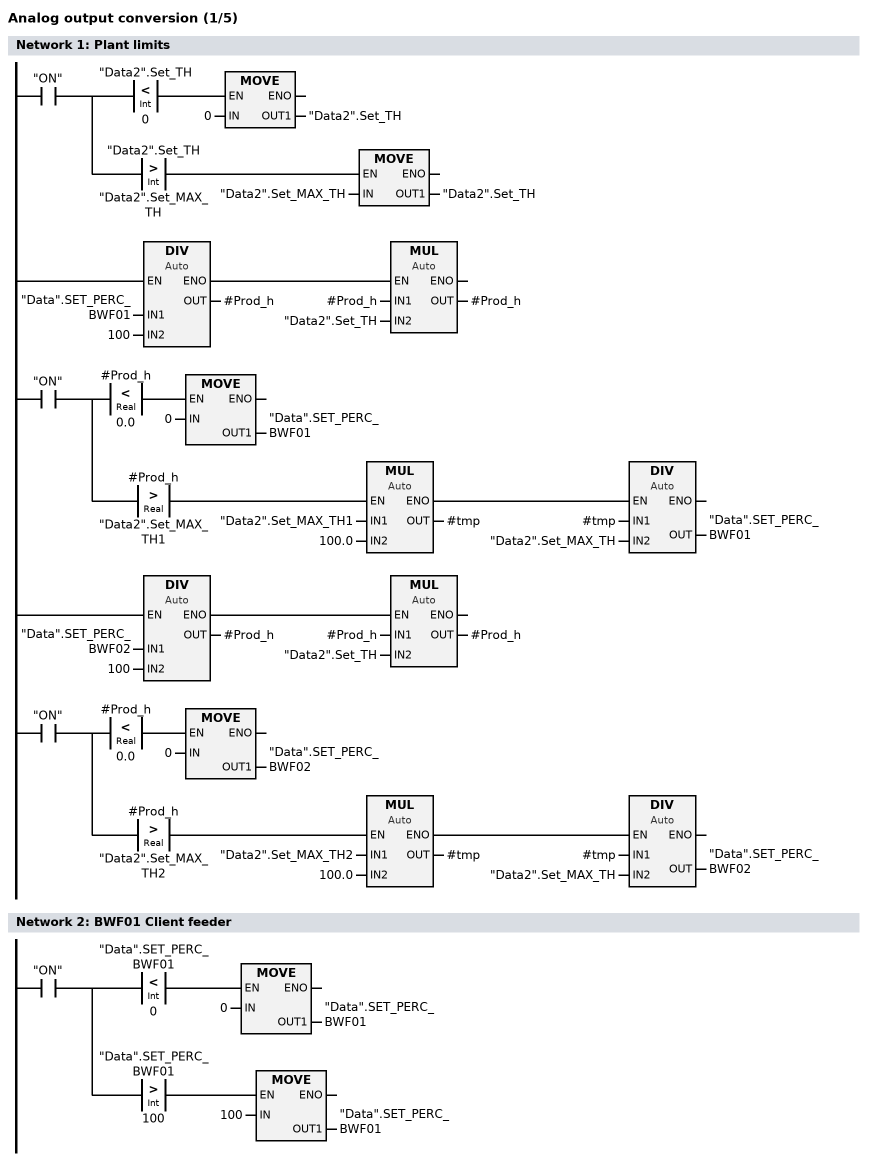
   RUNG wire#powerrail
      Contact( "ON" )
      wire#w1
      { S7_Templates := "SrcType := Int" } LT_Contact(in1 := "Data2".Set_TH, in2 := 0)
      { S7_GenerateENO := "TRUE" } Move(in := 0, out1 => "Data2".Set_TH)
   END_RUNG
   RUNG wire#w1
      { S7_Templates := "SrcType := Int" } GT_Contact(in1 := "Data2".Set_TH, in2 := "Data2".Set_MAX_TH)
      { S7_GenerateENO := "TRUE" } Move(in := "Data2".Set_MAX_TH, out1 => "Data2".Set_TH)
   END_RUNG
   RUNG wire#powerrail
      Div(in1 := "Data".SET_PERC_BWF01, in2 := 100, out => #Prod_h)
      Mul(in1 := #Prod_h, in2 := "Data2".Set_TH, out => #Prod_h)
   END_RUNG
   RUNG wire#powerrail
      Contact( "ON" )
      wire#w2
      { S7_Templates := "SrcType := Real" } LT_Contact(in1 := #Prod_h, in2 := 0.0)
      { S7_GenerateENO := "TRUE" } Move(in := 0, out1 => "Data".SET_PERC_BWF01)
   END_RUNG
   RUNG wire#w2
      { S7_Templates := "SrcType := Real" } GT_Contact(in1 := #Prod_h, in2 := "Data2".Set_MAX_TH1)
      Mul(in1 := "Data2".Set_MAX_TH1, in2 := 100.0, out => #tmp)
      Div(in1 := #tmp, in2 := "Data2".Set_MAX_TH, out => "Data".SET_PERC_BWF01)
   END_RUNG
   RUNG wire#powerrail
      Div(in1 := "Data".SET_PERC_BWF02, in2 := 100, out => #Prod_h)
      Mul(in1 := #Prod_h, in2 := "Data2".Set_TH, out => #Prod_h)
   END_RUNG
   RUNG wire#powerrail
      Contact( "ON" )
      wire#w3
      { S7_Templates := "SrcType := Real" } LT_Contact(in1 := #Prod_h, in2 := 0.0)
      { S7_GenerateENO := "TRUE" } Move(in := 0, out1 => "Data".SET_PERC_BWF02)
   END_RUNG
   RUNG wire#w3
      { S7_Templates := "SrcType := Real" } GT_Contact(in1 := #Prod_h, in2 := "Data2".Set_MAX_TH2)
      Mul(in1 := "Data2".Set_MAX_TH2, in2 := 100.0, out => #tmp)
      Div(in1 := #tmp, in2 := "Data2".Set_MAX_TH, out => "Data".SET_PERC_BWF02)
   END_RUNG
   // the same network as SCL:
   IF "ON" AND ("Data2".Set_TH < 0) THEN "Data2".Set_TH := 0; END_IF;
   IF "ON" AND ("Data2".Set_TH > "Data2".Set_MAX_TH) THEN "Data2".Set_TH := "Data2".Set_MAX_TH; END_IF;
   #Prod_h := "Data".SET_PERC_BWF01 / 100;
   #Prod_h := #Prod_h * "Data2".Set_TH;
   IF "ON" AND (#Prod_h < 0.0) THEN "Data".SET_PERC_BWF01 := 0; END_IF;
   IF "ON" AND (#Prod_h > "Data2".Set_MAX_TH1) THEN
       #tmp := "Data2".Set_MAX_TH1 * 100.0;
       "Data".SET_PERC_BWF01 := #tmp / "Data2".Set_MAX_TH;
   END_IF;
   #Prod_h := "Data".SET_PERC_BWF02 / 100;
   #Prod_h := #Prod_h * "Data2".Set_TH;
   IF "ON" AND (#Prod_h < 0.0) THEN "Data".SET_PERC_BWF02 := 0; END_IF;
   IF "ON" AND (#Prod_h > "Data2".Set_MAX_TH2) THEN
       #tmp := "Data2".Set_MAX_TH2 * 100.0;
       "Data".SET_PERC_BWF02 := #tmp / "Data2".Set_MAX_TH;
   END_IF;
END_REGION

REGION Network 2: BWF01 Client feeder
   RUNG wire#powerrail
      Contact( "ON" )
      wire#w1
      { S7_Templates := "SrcType := Int" } LT_Contact(in1 := "Data".SET_PERC_BWF01, in2 := 0)
      { S7_GenerateENO := "TRUE" } Move(in := 0, out1 => "Data".SET_PERC_BWF01)
   END_RUNG
   RUNG wire#w1
      { S7_Templates := "SrcType := Int" } GT_Contact(in1 := "Data".SET_PERC_BWF01, in2 := 100)
      { S7_GenerateENO := "TRUE" } Move(in := 100, out1 => "Data".SET_PERC_BWF01)
   END_RUNG
   // the same network as SCL:
   IF "ON" AND ("Data".SET_PERC_BWF01 < 0) THEN "Data".SET_PERC_BWF01 := 0; END_IF;
   IF "ON" AND ("Data".SET_PERC_BWF01 > 100) THEN "Data".SET_PERC_BWF01 := 100; END_IF;
END_REGION

REGION Network 3: BWF01 speed calculation
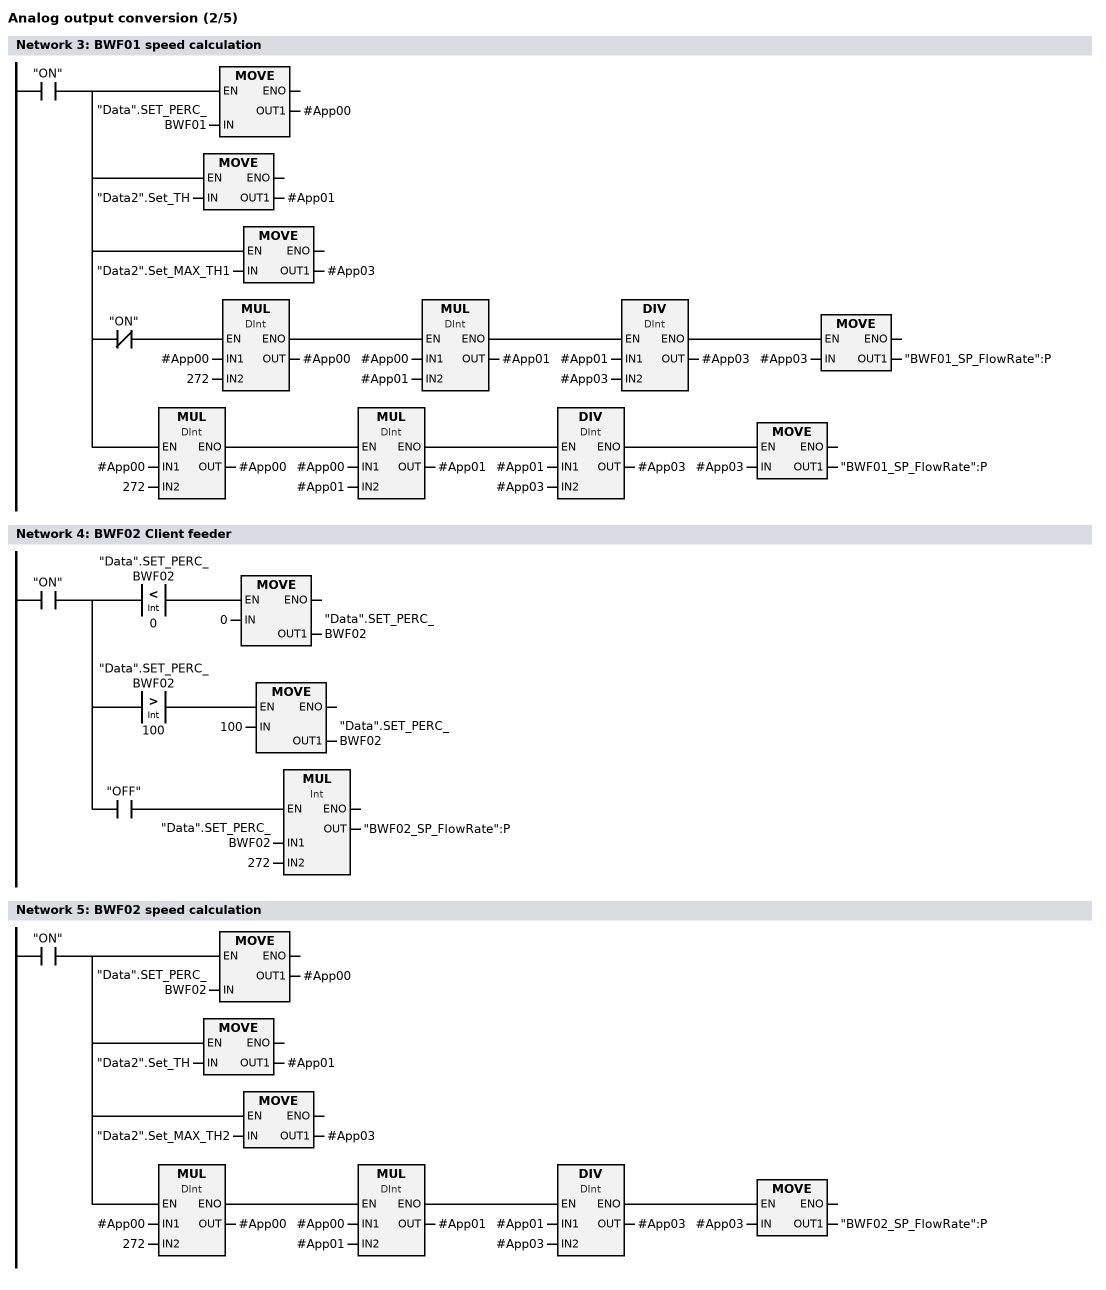
   RUNG wire#powerrail
      Contact( "ON" )
      wire#w1
      { S7_GenerateENO := "TRUE" } Move(in := "Data".SET_PERC_BWF01, out1 => #App00)
   END_RUNG
   RUNG wire#w1
      { S7_GenerateENO := "TRUE" } Move(in := "Data2".Set_TH, out1 => #App01)
   END_RUNG
   RUNG wire#w1
      { S7_GenerateENO := "TRUE" } Move(in := "Data2".Set_MAX_TH1, out1 => #App03)
   END_RUNG
   RUNG wire#w1
      I_Contact( "ON" )
      { S7_Templates := "SrcType := DInt"; S7_GenerateENO := "TRUE" } Mul(in1 := #App00, in2 := 272, out => #App00)
      { S7_Templates := "SrcType := DInt"; S7_GenerateENO := "TRUE" } Mul(in1 := #App00, in2 := #App01, out => #App01)
      { S7_Templates := "SrcType := DInt"; S7_GenerateENO := "TRUE" } Div(in1 := #App01, in2 := #App03, out => #App03)
      { S7_GenerateENO := "TRUE" } Move(in := #App03, out1 => "BWF01_SP_FlowRate":P)
   END_RUNG
   RUNG wire#w1
      { S7_Templates := "SrcType := DInt"; S7_GenerateENO := "TRUE" } Mul(in1 := #App00, in2 := 272, out => #App00)
      { S7_Templates := "SrcType := DInt"; S7_GenerateENO := "TRUE" } Mul(in1 := #App00, in2 := #App01, out => #App01)
      { S7_Templates := "SrcType := DInt"; S7_GenerateENO := "TRUE" } Div(in1 := #App01, in2 := #App03, out => #App03)
      { S7_GenerateENO := "TRUE" } Move(in := #App03, out1 => "BWF01_SP_FlowRate":P)
   END_RUNG
   // the same network as SCL:
   // ENO of a box is taken as its EN; it also drops when the box reports an error
   IF "ON" THEN
       #App00 := "Data".SET_PERC_BWF01;
       #App01 := "Data2".Set_TH;
       #App03 := "Data2".Set_MAX_TH1;
   END_IF;
   IF "ON" AND NOT "ON" THEN
       #App00 := #App00 * 272;
       #App01 := #App00 * #App01;
       #App03 := #App01 / #App03;
       "BWF01_SP_FlowRate":P := #App03;
   END_IF;
   IF "ON" THEN
       #App00 := #App00 * 272;
       #App01 := #App00 * #App01;
       #App03 := #App01 / #App03;
       "BWF01_SP_FlowRate":P := #App03;
   END_IF;
END_REGION

REGION Network 4: BWF02 Client feeder
   RUNG wire#powerrail
      Contact( "ON" )
      wire#w1
      { S7_Templates := "SrcType := Int" } LT_Contact(in1 := "Data".SET_PERC_BWF02, in2 := 0)
      { S7_GenerateENO := "TRUE" } Move(in := 0, out1 => "Data".SET_PERC_BWF02)
   END_RUNG
   RUNG wire#w1
      { S7_Templates := "SrcType := Int" } GT_Contact(in1 := "Data".SET_PERC_BWF02, in2 := 100)
      { S7_GenerateENO := "TRUE" } Move(in := 100, out1 => "Data".SET_PERC_BWF02)
   END_RUNG
   RUNG wire#w1
      Contact( "OFF" )
      { S7_Templates := "SrcType := Int"; S7_GenerateENO := "TRUE" } Mul(in1 := "Data".SET_PERC_BWF02, in2 := 272, out => "BWF02_SP_FlowRate":P)
   END_RUNG
   // the same network as SCL:
   IF "ON" AND ("Data".SET_PERC_BWF02 < 0) THEN "Data".SET_PERC_BWF02 := 0; END_IF;
   IF "ON" AND ("Data".SET_PERC_BWF02 > 100) THEN "Data".SET_PERC_BWF02 := 100; END_IF;
   IF "ON" AND "OFF" THEN "BWF02_SP_FlowRate":P := "Data".SET_PERC_BWF02 * 272; END_IF;
END_REGION

REGION Network 5: BWF02 speed calculation
   RUNG wire#powerrail
      Contact( "ON" )
      wire#w1
      { S7_GenerateENO := "TRUE" } Move(in := "Data".SET_PERC_BWF02, out1 => #App00)
   END_RUNG
   RUNG wire#w1
      { S7_GenerateENO := "TRUE" } Move(in := "Data2".Set_TH, out1 => #App01)
   END_RUNG
   RUNG wire#w1
      { S7_GenerateENO := "TRUE" } Move(in := "Data2".Set_MAX_TH2, out1 => #App03)
   END_RUNG
   RUNG wire#w1
      { S7_Templates := "SrcType := DInt"; S7_GenerateENO := "TRUE" } Mul(in1 := #App00, in2 := 272, out => #App00)
      { S7_Templates := "SrcType := DInt"; S7_GenerateENO := "TRUE" } Mul(in1 := #App00, in2 := #App01, out => #App01)
      { S7_Templates := "SrcType := DInt"; S7_GenerateENO := "TRUE" } Div(in1 := #App01, in2 := #App03, out => #App03)
      { S7_GenerateENO := "TRUE" } Move(in := #App03, out1 => "BWF02_SP_FlowRate":P)
   END_RUNG
   // the same network as SCL:
   // ENO of a box is taken as its EN; it also drops when the box reports an error
   IF "ON" THEN
       #App00 := "Data".SET_PERC_BWF02;
       #App01 := "Data2".Set_TH;
       #App03 := "Data2".Set_MAX_TH2;
       #App00 := #App00 * 272;
       #App01 := #App00 * #App01;
       #App03 := #App01 / #App03;
       "BWF02_SP_FlowRate":P := #App03;
   END_IF;
END_REGION

REGION Network 6: RD-01 Cylinder
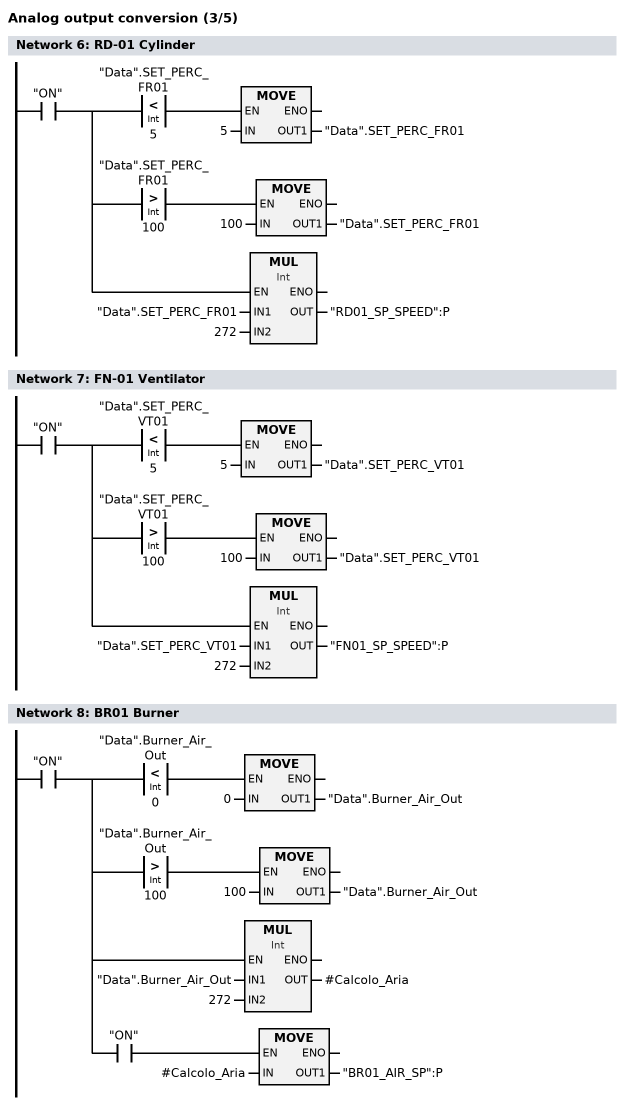
   RUNG wire#powerrail
      Contact( "ON" )
      wire#w1
      { S7_Templates := "SrcType := Int" } LT_Contact(in1 := "Data".SET_PERC_FR01, in2 := 5)
      { S7_GenerateENO := "TRUE" } Move(in := 5, out1 => "Data".SET_PERC_FR01)
   END_RUNG
   RUNG wire#w1
      { S7_Templates := "SrcType := Int" } GT_Contact(in1 := "Data".SET_PERC_FR01, in2 := 100)
      { S7_GenerateENO := "TRUE" } Move(in := 100, out1 => "Data".SET_PERC_FR01)
   END_RUNG
   RUNG wire#w1
      { S7_Templates := "SrcType := Int"; S7_GenerateENO := "TRUE" } Mul(in1 := "Data".SET_PERC_FR01, in2 := 272, out => "RD01_SP_SPEED":P)
   END_RUNG
   // the same network as SCL:
   IF "ON" AND ("Data".SET_PERC_FR01 < 5) THEN "Data".SET_PERC_FR01 := 5; END_IF;
   IF "ON" AND ("Data".SET_PERC_FR01 > 100) THEN "Data".SET_PERC_FR01 := 100; END_IF;
   IF "ON" THEN "RD01_SP_SPEED":P := "Data".SET_PERC_FR01 * 272; END_IF;
END_REGION

REGION Network 7: FN-01 Ventilator
   RUNG wire#powerrail
      Contact( "ON" )
      wire#w1
      { S7_Templates := "SrcType := Int" } LT_Contact(in1 := "Data".SET_PERC_VT01, in2 := 5)
      { S7_GenerateENO := "TRUE" } Move(in := 5, out1 => "Data".SET_PERC_VT01)
   END_RUNG
   RUNG wire#w1
      { S7_Templates := "SrcType := Int" } GT_Contact(in1 := "Data".SET_PERC_VT01, in2 := 100)
      { S7_GenerateENO := "TRUE" } Move(in := 100, out1 => "Data".SET_PERC_VT01)
   END_RUNG
   RUNG wire#w1
      { S7_Templates := "SrcType := Int"; S7_GenerateENO := "TRUE" } Mul(in1 := "Data".SET_PERC_VT01, in2 := 272, out => "FN01_SP_SPEED":P)
   END_RUNG
   // the same network as SCL:
   IF "ON" AND ("Data".SET_PERC_VT01 < 5) THEN "Data".SET_PERC_VT01 := 5; END_IF;
   IF "ON" AND ("Data".SET_PERC_VT01 > 100) THEN "Data".SET_PERC_VT01 := 100; END_IF;
   IF "ON" THEN "FN01_SP_SPEED":P := "Data".SET_PERC_VT01 * 272; END_IF;
END_REGION

REGION Network 8: BR01 Burner
   RUNG wire#powerrail
      Contact( "ON" )
      wire#w1
      { S7_Templates := "SrcType := Int" } LT_Contact(in1 := "Data".Burner_Air_Out, in2 := 0)
      { S7_GenerateENO := "TRUE" } Move(in := 0, out1 => "Data".Burner_Air_Out)
   END_RUNG
   RUNG wire#w1
      { S7_Templates := "SrcType := Int" } GT_Contact(in1 := "Data".Burner_Air_Out, in2 := 100)
      { S7_GenerateENO := "TRUE" } Move(in := 100, out1 => "Data".Burner_Air_Out)
   END_RUNG
   RUNG wire#w1
      { S7_Templates := "SrcType := Int"; S7_GenerateENO := "TRUE" } Mul(in1 := "Data".Burner_Air_Out, in2 := 272, out => #Calcolo_Aria)
   END_RUNG
   RUNG wire#w1
      Contact( "ON" )
      { S7_GenerateENO := "TRUE" } Move(in := #Calcolo_Aria, out1 => "BR01_AIR_SP":P)
   END_RUNG
   // the same network as SCL:
   IF "ON" AND ("Data".Burner_Air_Out < 0) THEN "Data".Burner_Air_Out := 0; END_IF;
   IF "ON" AND ("Data".Burner_Air_Out > 100) THEN "Data".Burner_Air_Out := 100; END_IF;
   IF "ON" THEN #Calcolo_Aria := "Data".Burner_Air_Out * 272; END_IF;
   IF "ON" AND "ON" THEN "BR01_AIR_SP":P := #Calcolo_Aria; END_IF;
END_REGION

REGION Network 9: BR01 Burner - Gas
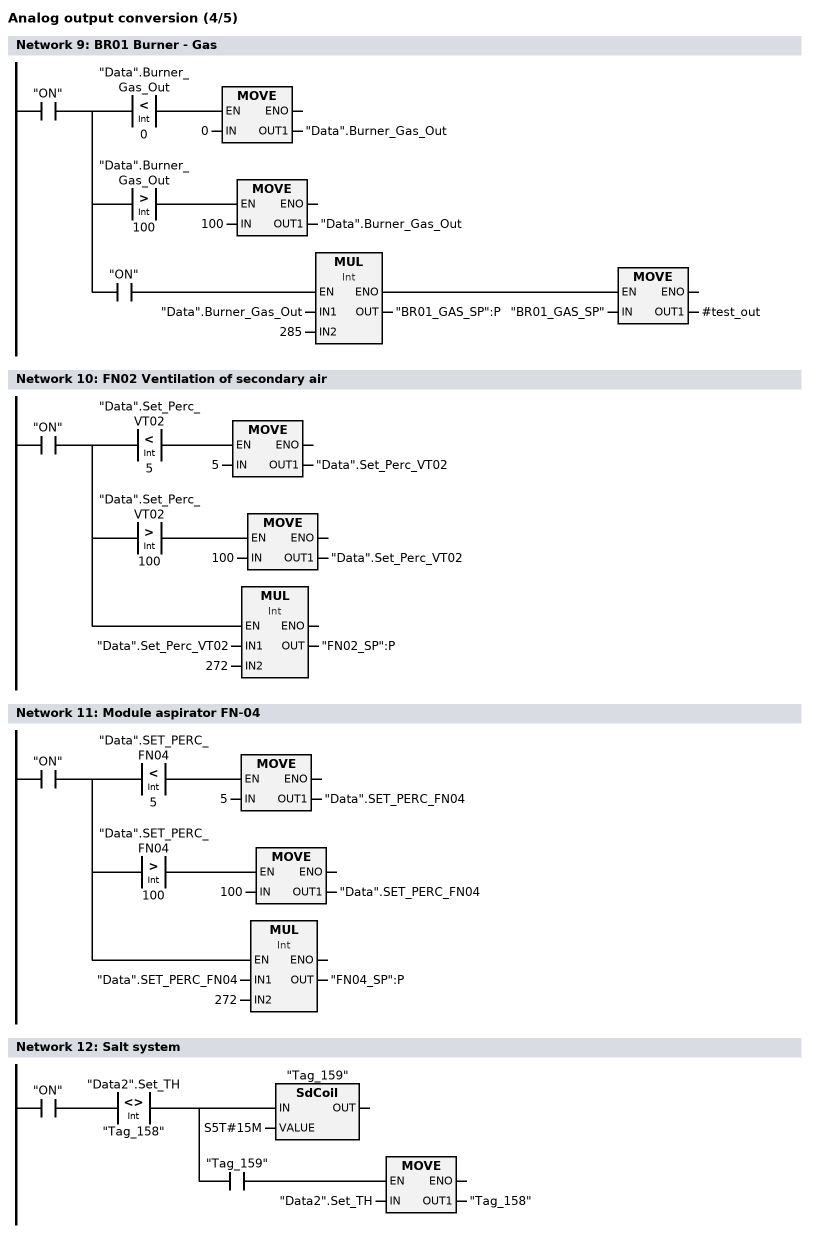
   RUNG wire#powerrail
      Contact( "ON" )
      wire#w1
      { S7_Templates := "SrcType := Int" } LT_Contact(in1 := "Data".Burner_Gas_Out, in2 := 0)
      { S7_GenerateENO := "TRUE" } Move(in := 0, out1 => "Data".Burner_Gas_Out)
   END_RUNG
   RUNG wire#w1
      { S7_Templates := "SrcType := Int" } GT_Contact(in1 := "Data".Burner_Gas_Out, in2 := 100)
      { S7_GenerateENO := "TRUE" } Move(in := 100, out1 => "Data".Burner_Gas_Out)
   END_RUNG
   RUNG wire#w1
      Contact( "ON" )
      { S7_Templates := "SrcType := Int"; S7_GenerateENO := "TRUE" } Mul(in1 := "Data".Burner_Gas_Out, in2 := 285, out => "BR01_GAS_SP":P)
      Move(in := "BR01_GAS_SP", out1 => #test_out)
   END_RUNG
   // the same network as SCL:
   // ENO of a box is taken as its EN; it also drops when the box reports an error
   IF "ON" AND ("Data".Burner_Gas_Out < 0) THEN "Data".Burner_Gas_Out := 0; END_IF;
   IF "ON" AND ("Data".Burner_Gas_Out > 100) THEN "Data".Burner_Gas_Out := 100; END_IF;
   IF "ON" AND "ON" THEN
       "BR01_GAS_SP":P := "Data".Burner_Gas_Out * 285;
       #test_out := "BR01_GAS_SP";
   END_IF;
END_REGION

REGION Network 10: FN02 Ventilation of secondary air
   RUNG wire#powerrail
      Contact( "ON" )
      wire#w1
      { S7_Templates := "SrcType := Int" } LT_Contact(in1 := "Data".Set_Perc_VT02, in2 := 5)
      { S7_GenerateENO := "TRUE" } Move(in := 5, out1 => "Data".Set_Perc_VT02)
   END_RUNG
   RUNG wire#w1
      { S7_Templates := "SrcType := Int" } GT_Contact(in1 := "Data".Set_Perc_VT02, in2 := 100)
      { S7_GenerateENO := "TRUE" } Move(in := 100, out1 => "Data".Set_Perc_VT02)
   END_RUNG
   RUNG wire#w1
      { S7_Templates := "SrcType := Int"; S7_GenerateENO := "TRUE" } Mul(in1 := "Data".Set_Perc_VT02, in2 := 272, out => "FN02_SP":P)
   END_RUNG
   // the same network as SCL:
   IF "ON" AND ("Data".Set_Perc_VT02 < 5) THEN "Data".Set_Perc_VT02 := 5; END_IF;
   IF "ON" AND ("Data".Set_Perc_VT02 > 100) THEN "Data".Set_Perc_VT02 := 100; END_IF;
   IF "ON" THEN "FN02_SP":P := "Data".Set_Perc_VT02 * 272; END_IF;
END_REGION

REGION Network 11: Module aspirator FN-04
   RUNG wire#powerrail
      Contact( "ON" )
      wire#w1
      { S7_Templates := "SrcType := Int" } LT_Contact(in1 := "Data".SET_PERC_FN04, in2 := 5)
      { S7_GenerateENO := "TRUE" } Move(in := 5, out1 => "Data".SET_PERC_FN04)
   END_RUNG
   RUNG wire#w1
      { S7_Templates := "SrcType := Int" } GT_Contact(in1 := "Data".SET_PERC_FN04, in2 := 100)
      { S7_GenerateENO := "TRUE" } Move(in := 100, out1 => "Data".SET_PERC_FN04)
   END_RUNG
   RUNG wire#w1
      { S7_Templates := "SrcType := Int"; S7_GenerateENO := "TRUE" } Mul(in1 := "Data".SET_PERC_FN04, in2 := 272, out => "FN04_SP":P)
   END_RUNG
   // the same network as SCL:
   IF "ON" AND ("Data".SET_PERC_FN04 < 5) THEN "Data".SET_PERC_FN04 := 5; END_IF;
   IF "ON" AND ("Data".SET_PERC_FN04 > 100) THEN "Data".SET_PERC_FN04 := 100; END_IF;
   IF "ON" THEN "FN04_SP":P := "Data".SET_PERC_FN04 * 272; END_IF;
END_REGION

REGION Network 12: Salt system
   // no SCL statement known for SdCoil: written as a call
   #_w1 := "ON" AND ("Data2".Set_TH <> "Tag_158");
   SdCoil(in := #_w1, value := S5T#15M, operand := "Tag_159");
   IF #_w1 AND "Tag_159" THEN "Tag_158" := "Data2".Set_TH; END_IF;
END_REGION

REGION Network 13: Send output to perifery
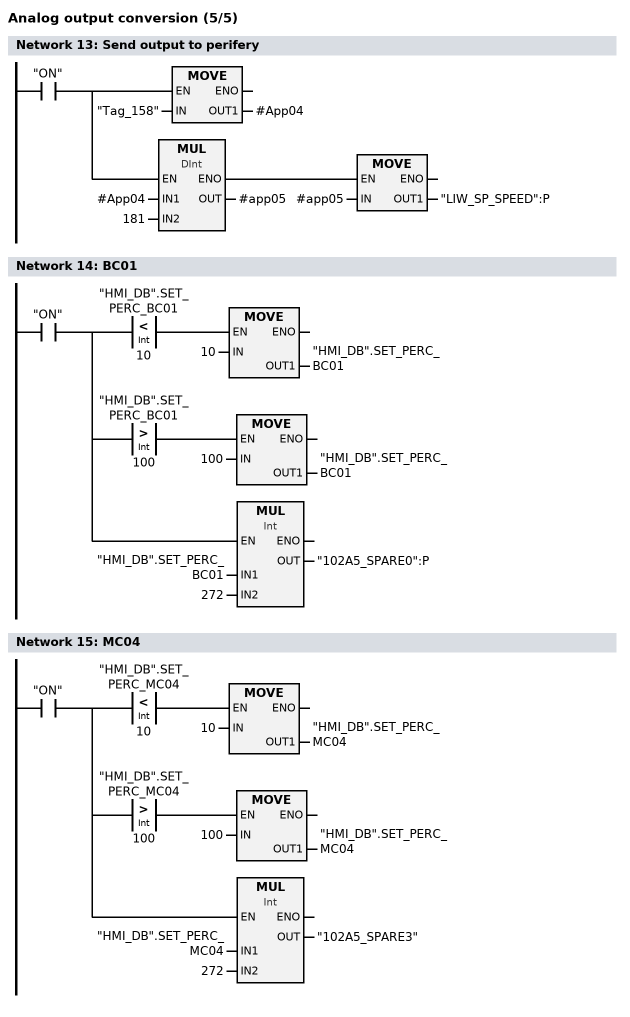
   RUNG wire#powerrail
      Contact( "ON" )
      wire#w1
      { S7_GenerateENO := "TRUE" } Move(in := "Tag_158", out1 => #App04)
   END_RUNG
   RUNG wire#w1
      { S7_Templates := "SrcType := DInt"; S7_GenerateENO := "TRUE" } Mul(in1 := #App04, in2 := 181, out => #app05)
      { S7_GenerateENO := "TRUE" } Move(in := #app05, out1 => "LIW_SP_SPEED":P)
   END_RUNG
   // the same network as SCL:
   // ENO of a box is taken as its EN; it also drops when the box reports an error
   IF "ON" THEN
       #App04 := "Tag_158";
       #app05 := #App04 * 181;
       "LIW_SP_SPEED":P := #app05;
   END_IF;
END_REGION

REGION Network 14: BC01
   RUNG wire#powerrail
      Contact( "ON" )
      wire#w1
      { S7_Templates := "SrcType := Int" } LT_Contact(in1 := "HMI_DB".SET_PERC_BC01, in2 := 10)
      { S7_GenerateENO := "TRUE" } Move(in := 10, out1 => "HMI_DB".SET_PERC_BC01)
   END_RUNG
   RUNG wire#w1
      { S7_Templates := "SrcType := Int" } GT_Contact(in1 := "HMI_DB".SET_PERC_BC01, in2 := 100)
      { S7_GenerateENO := "TRUE" } Move(in := 100, out1 => "HMI_DB".SET_PERC_BC01)
   END_RUNG
   RUNG wire#w1
      { S7_Templates := "SrcType := Int"; S7_GenerateENO := "TRUE" } Mul(in1 := "HMI_DB".SET_PERC_BC01, in2 := 272, out => "102A5_SPARE0":P)
   END_RUNG
   // the same network as SCL:
   IF "ON" AND ("HMI_DB".SET_PERC_BC01 < 10) THEN "HMI_DB".SET_PERC_BC01 := 10; END_IF;
   IF "ON" AND ("HMI_DB".SET_PERC_BC01 > 100) THEN "HMI_DB".SET_PERC_BC01 := 100; END_IF;
   IF "ON" THEN "102A5_SPARE0":P := "HMI_DB".SET_PERC_BC01 * 272; END_IF;
END_REGION

REGION Network 15: MC04
   RUNG wire#powerrail
      Contact( "ON" )
      wire#w1
      { S7_Templates := "SrcType := Int" } LT_Contact(in1 := "HMI_DB".SET_PERC_MC04, in2 := 10)
      { S7_GenerateENO := "TRUE" } Move(in := 10, out1 => "HMI_DB".SET_PERC_MC04)
   END_RUNG
   RUNG wire#w1
      { S7_Templates := "SrcType := Int" } GT_Contact(in1 := "HMI_DB".SET_PERC_MC04, in2 := 100)
      { S7_GenerateENO := "TRUE" } Move(in := 100, out1 => "HMI_DB".SET_PERC_MC04)
   END_RUNG
   RUNG wire#w1
      { S7_Templates := "SrcType := Int"; S7_GenerateENO := "TRUE" } Mul(in1 := "HMI_DB".SET_PERC_MC04, in2 := 272, out => "102A5_SPARE3")
   END_RUNG
   // the same network as SCL:
   IF "ON" AND ("HMI_DB".SET_PERC_MC04 < 10) THEN "HMI_DB".SET_PERC_MC04 := 10; END_IF;
   IF "ON" AND ("HMI_DB".SET_PERC_MC04 > 100) THEN "HMI_DB".SET_PERC_MC04 := 100; END_IF;
   IF "ON" THEN "102A5_SPARE3" := "HMI_DB".SET_PERC_MC04 * 272; END_IF;
END_REGION
END_FUNCTION

FUNCTION "Simulation" : Void   // FC20, LAD
{ S7_Optimized_Access := 'TRUE' }
VERSION : 0.1
   VAR_TEMP
      BuffInc : Int;
   END_VAR
BEGIN

REGION Network 1
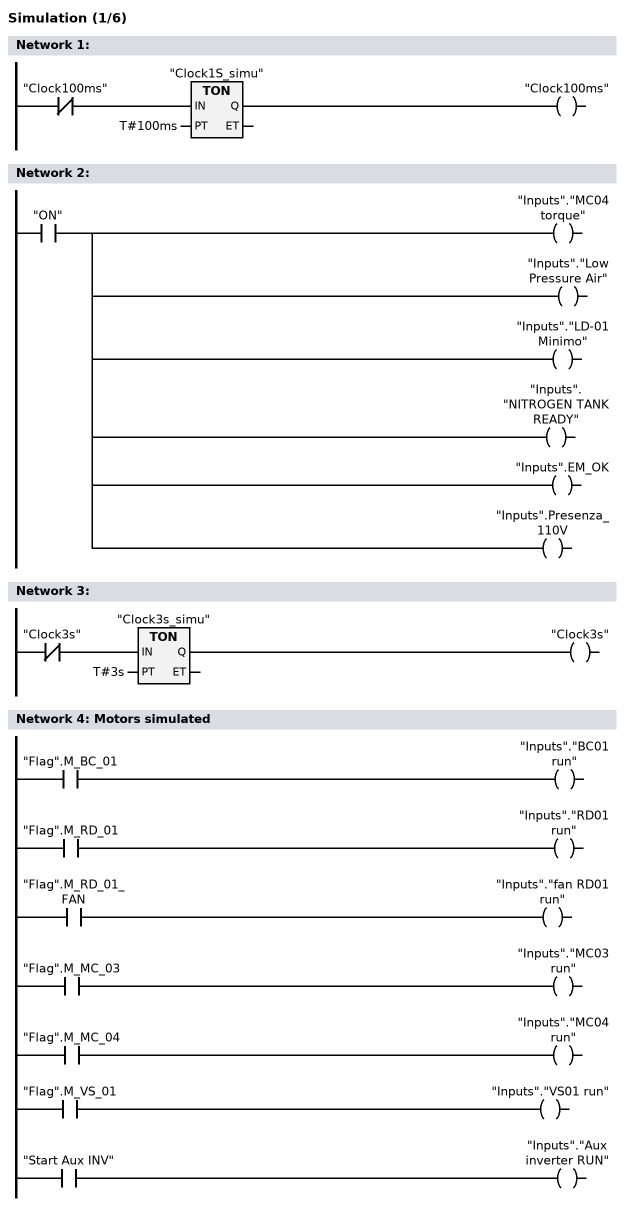
   "Clock1S_simu".TON(IN := NOT "Clock100ms", PT := T#100ms);
   "Clock100ms" := "Clock1S_simu".Q;
END_REGION

REGION Network 2
   RUNG wire#powerrail
      Contact( "ON" )
      wire#w1
      Coil( "Inputs"."MC04 torque" )
   END_RUNG
   RUNG wire#w1
      Coil( "Inputs"."Low Pressure Air" )
   END_RUNG
   RUNG wire#w1
      Coil( "Inputs"."LD-01 Minimo" )
   END_RUNG
   RUNG wire#w1
      Coil( "Inputs"."NITROGEN TANK READY" )
   END_RUNG
   RUNG wire#w1
      Coil( "Inputs".EM_OK )
   END_RUNG
   RUNG wire#w1
      Coil( "Inputs".Presenza_110V )
   END_RUNG
   // the same network as SCL:
   "Inputs"."MC04 torque" := "ON";
   "Inputs"."Low Pressure Air" := "ON";
   "Inputs"."LD-01 Minimo" := "ON";
   "Inputs"."NITROGEN TANK READY" := "ON";
   "Inputs".EM_OK := "ON";
   "Inputs".Presenza_110V := "ON";
END_REGION

REGION Network 3
   "Clock3s_simu".TON(IN := NOT "Clock3s", PT := T#3s);
   "Clock3s" := "Clock3s_simu".Q;
END_REGION

REGION Network 4: Motors simulated
   RUNG wire#powerrail
      Contact( "Flag".M_BC_01 )
      Coil( "Inputs"."BC01 run" )
   END_RUNG
   RUNG wire#powerrail
      Contact( "Flag".M_RD_01 )
      Coil( "Inputs"."RD01 run" )
   END_RUNG
   RUNG wire#powerrail
      Contact( "Flag".M_RD_01_FAN )
      Coil( "Inputs"."fan RD01 run" )
   END_RUNG
   RUNG wire#powerrail
      Contact( "Flag".M_MC_03 )
      Coil( "Inputs"."MC03 run" )
   END_RUNG
   RUNG wire#powerrail
      Contact( "Flag".M_MC_04 )
      Coil( "Inputs"."MC04 run" )
   END_RUNG
   RUNG wire#powerrail
      Contact( "Flag".M_VS_01 )
      Coil( "Inputs"."VS01 run" )
   END_RUNG
   RUNG wire#powerrail
      Contact( "Start Aux INV" )
      Coil( "Inputs"."Aux inverter RUN" )
   END_RUNG
   // the same network as SCL:
   "Inputs"."BC01 run" := "Flag".M_BC_01;
   "Inputs"."RD01 run" := "Flag".M_RD_01;
   "Inputs"."fan RD01 run" := "Flag".M_RD_01_FAN;
   "Inputs"."MC03 run" := "Flag".M_MC_03;
   "Inputs"."MC04 run" := "Flag".M_MC_04;
   "Inputs"."VS01 run" := "Flag".M_VS_01;
   "Inputs"."Aux inverter RUN" := "Start Aux INV";
END_REGION

REGION Network 5: MV
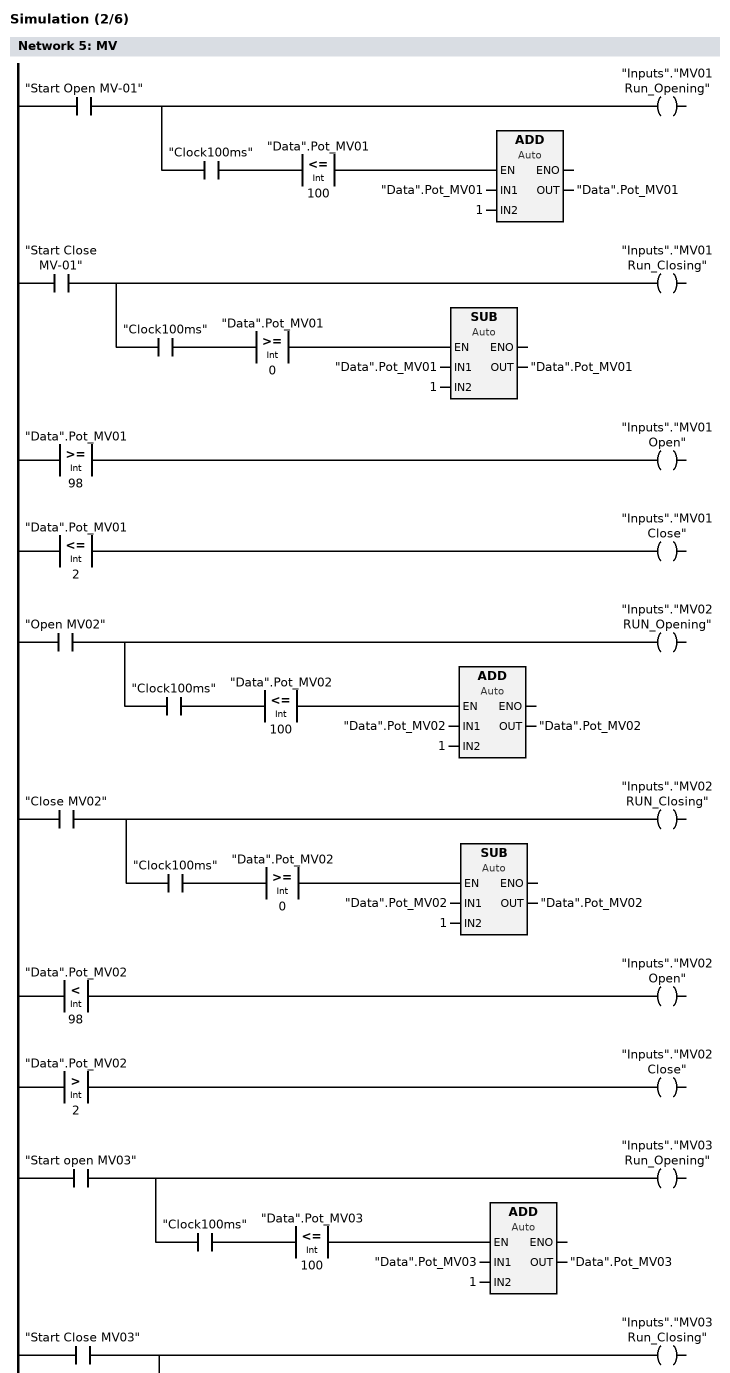
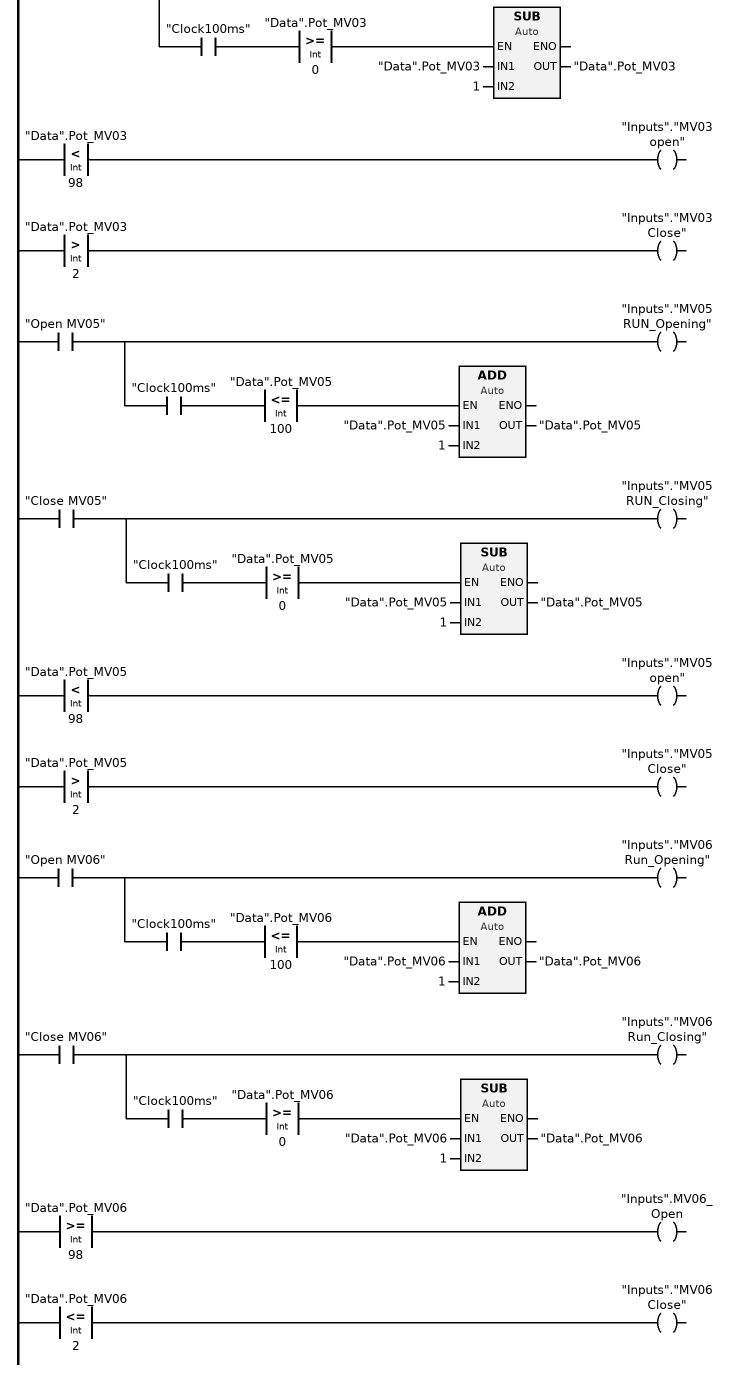
   RUNG wire#powerrail
      Contact( "Start Open MV-01" )
      wire#w1
      Coil( "Inputs"."MV01 Run_Opening" )
   END_RUNG
   RUNG wire#w1
      Contact( "Clock100ms" )
      { S7_Templates := "SrcType := Int" } LE_Contact(in1 := "Data".Pot_MV01, in2 := 100)
      Add(in1 := "Data".Pot_MV01, in2 := 1, out => "Data".Pot_MV01)
   END_RUNG
   RUNG wire#powerrail
      Contact( "Start Close MV-01" )
      wire#w2
      Coil( "Inputs"."MV01 Run_Closing" )
   END_RUNG
   RUNG wire#w2
      Contact( "Clock100ms" )
      { S7_Templates := "SrcType := Int" } GE_Contact(in1 := "Data".Pot_MV01, in2 := 0)
      Sub(in1 := "Data".Pot_MV01, in2 := 1, out => "Data".Pot_MV01)
   END_RUNG
   RUNG wire#powerrail
      { S7_Templates := "SrcType := Int" } GE_Contact(in1 := "Data".Pot_MV01, in2 := 98)
      Coil( "Inputs"."MV01 Open" )
   END_RUNG
   RUNG wire#powerrail
      { S7_Templates := "SrcType := Int" } LE_Contact(in1 := "Data".Pot_MV01, in2 := 2)
      Coil( "Inputs"."MV01 Close" )
   END_RUNG
   RUNG wire#powerrail
      Contact( "Open MV02" )
      wire#w3
      Coil( "Inputs"."MV02 RUN_Opening" )
   END_RUNG
   RUNG wire#w3
      Contact( "Clock100ms" )
      { S7_Templates := "SrcType := Int" } LE_Contact(in1 := "Data".Pot_MV02, in2 := 100)
      Add(in1 := "Data".Pot_MV02, in2 := 1, out => "Data".Pot_MV02)
   END_RUNG
   RUNG wire#powerrail
      Contact( "Close MV02" )
      wire#w4
      Coil( "Inputs"."MV02 RUN_Closing" )
   END_RUNG
   RUNG wire#w4
      Contact( "Clock100ms" )
      { S7_Templates := "SrcType := Int" } GE_Contact(in1 := "Data".Pot_MV02, in2 := 0)
      Sub(in1 := "Data".Pot_MV02, in2 := 1, out => "Data".Pot_MV02)
   END_RUNG
   RUNG wire#powerrail
      { S7_Templates := "SrcType := Int" } LT_Contact(in1 := "Data".Pot_MV02, in2 := 98)
      Coil( "Inputs"."MV02 Open" )
   END_RUNG
   RUNG wire#powerrail
      { S7_Templates := "SrcType := Int" } GT_Contact(in1 := "Data".Pot_MV02, in2 := 2)
      Coil( "Inputs"."MV02 Close" )
   END_RUNG
   RUNG wire#powerrail
      Contact( "Start open MV03" )
      wire#w5
      Coil( "Inputs"."MV03 Run_Opening" )
   END_RUNG
   RUNG wire#w5
      Contact( "Clock100ms" )
      { S7_Templates := "SrcType := Int" } LE_Contact(in1 := "Data".Pot_MV03, in2 := 100)
      Add(in1 := "Data".Pot_MV03, in2 := 1, out => "Data".Pot_MV03)
   END_RUNG
   RUNG wire#powerrail
      Contact( "Start Close MV03" )
      wire#w6
      Coil( "Inputs"."MV03 Run_Closing" )
   END_RUNG
   RUNG wire#w6
      Contact( "Clock100ms" )
      { S7_Templates := "SrcType := Int" } GE_Contact(in1 := "Data".Pot_MV03, in2 := 0)
      Sub(in1 := "Data".Pot_MV03, in2 := 1, out => "Data".Pot_MV03)
   END_RUNG
   RUNG wire#powerrail
      { S7_Templates := "SrcType := Int" } LT_Contact(in1 := "Data".Pot_MV03, in2 := 98)
      Coil( "Inputs"."MV03 open" )
   END_RUNG
   RUNG wire#powerrail
      { S7_Templates := "SrcType := Int" } GT_Contact(in1 := "Data".Pot_MV03, in2 := 2)
      Coil( "Inputs"."MV03 Close" )
   END_RUNG
   RUNG wire#powerrail
      Contact( "Open MV05" )
      wire#w7
      Coil( "Inputs"."MV05 RUN_Opening" )
   END_RUNG
   RUNG wire#w7
      Contact( "Clock100ms" )
      { S7_Templates := "SrcType := Int" } LE_Contact(in1 := "Data".Pot_MV05, in2 := 100)
      Add(in1 := "Data".Pot_MV05, in2 := 1, out => "Data".Pot_MV05)
   END_RUNG
   RUNG wire#powerrail
      Contact( "Close MV05" )
      wire#w8
      Coil( "Inputs"."MV05 RUN_Closing" )
   END_RUNG
   RUNG wire#w8
      Contact( "Clock100ms" )
      { S7_Templates := "SrcType := Int" } GE_Contact(in1 := "Data".Pot_MV05, in2 := 0)
      Sub(in1 := "Data".Pot_MV05, in2 := 1, out => "Data".Pot_MV05)
   END_RUNG
   RUNG wire#powerrail
      { S7_Templates := "SrcType := Int" } LT_Contact(in1 := "Data".Pot_MV05, in2 := 98)
      Coil( "Inputs"."MV05 open" )
   END_RUNG
   RUNG wire#powerrail
      { S7_Templates := "SrcType := Int" } GT_Contact(in1 := "Data".Pot_MV05, in2 := 2)
      Coil( "Inputs"."MV05 Close" )
   END_RUNG
   RUNG wire#powerrail
      Contact( "Open MV06" )
      wire#w9
      Coil( "Inputs"."MV06 Run_Opening" )
   END_RUNG
   RUNG wire#w9
      Contact( "Clock100ms" )
      { S7_Templates := "SrcType := Int" } LE_Contact(in1 := "Data".Pot_MV06, in2 := 100)
      Add(in1 := "Data".Pot_MV06, in2 := 1, out => "Data".Pot_MV06)
   END_RUNG
   RUNG wire#powerrail
      Contact( "Close MV06" )
      wire#w10
      Coil( "Inputs"."MV06 Run_Closing" )
   END_RUNG
   RUNG wire#w10
      Contact( "Clock100ms" )
      { S7_Templates := "SrcType := Int" } GE_Contact(in1 := "Data".Pot_MV06, in2 := 0)
      Sub(in1 := "Data".Pot_MV06, in2 := 1, out => "Data".Pot_MV06)
   END_RUNG
   RUNG wire#powerrail
      { S7_Templates := "SrcType := Int" } GE_Contact(in1 := "Data".Pot_MV06, in2 := 98)
      Coil( "Inputs".MV06_Open )
   END_RUNG
   RUNG wire#powerrail
      { S7_Templates := "SrcType := Int" } LE_Contact(in1 := "Data".Pot_MV06, in2 := 2)
      Coil( "Inputs"."MV06 Close" )
   END_RUNG
   // the same network as SCL:
   "Inputs"."MV01 Run_Opening" := "Start Open MV-01";
   IF "Start Open MV-01" AND "Clock100ms" AND ("Data".Pot_MV01 <= 100) THEN
       "Data".Pot_MV01 := "Data".Pot_MV01 + 1;
   END_IF;
   "Inputs"."MV01 Run_Closing" := "Start Close MV-01";
   IF "Start Close MV-01" AND "Clock100ms" AND ("Data".Pot_MV01 >= 0) THEN
       "Data".Pot_MV01 := "Data".Pot_MV01 - 1;
   END_IF;
   "Inputs"."MV01 Open" := "Data".Pot_MV01 >= 98;
   "Inputs"."MV01 Close" := "Data".Pot_MV01 <= 2;
   "Inputs"."MV02 RUN_Opening" := "Open MV02";
   IF "Open MV02" AND "Clock100ms" AND ("Data".Pot_MV02 <= 100) THEN
       "Data".Pot_MV02 := "Data".Pot_MV02 + 1;
   END_IF;
   "Inputs"."MV02 RUN_Closing" := "Close MV02";
   IF "Close MV02" AND "Clock100ms" AND ("Data".Pot_MV02 >= 0) THEN
       "Data".Pot_MV02 := "Data".Pot_MV02 - 1;
   END_IF;
   "Inputs"."MV02 Open" := "Data".Pot_MV02 < 98;
   "Inputs"."MV02 Close" := "Data".Pot_MV02 > 2;
   "Inputs"."MV03 Run_Opening" := "Start open MV03";
   IF "Start open MV03" AND "Clock100ms" AND ("Data".Pot_MV03 <= 100) THEN
       "Data".Pot_MV03 := "Data".Pot_MV03 + 1;
   END_IF;
   "Inputs"."MV03 Run_Closing" := "Start Close MV03";
   IF "Start Close MV03" AND "Clock100ms" AND ("Data".Pot_MV03 >= 0) THEN
       "Data".Pot_MV03 := "Data".Pot_MV03 - 1;
   END_IF;
   "Inputs"."MV03 open" := "Data".Pot_MV03 < 98;
   "Inputs"."MV03 Close" := "Data".Pot_MV03 > 2;
   "Inputs"."MV05 RUN_Opening" := "Open MV05";
   IF "Open MV05" AND "Clock100ms" AND ("Data".Pot_MV05 <= 100) THEN
       "Data".Pot_MV05 := "Data".Pot_MV05 + 1;
   END_IF;
   "Inputs"."MV05 RUN_Closing" := "Close MV05";
   IF "Close MV05" AND "Clock100ms" AND ("Data".Pot_MV05 >= 0) THEN
       "Data".Pot_MV05 := "Data".Pot_MV05 - 1;
   END_IF;
   "Inputs"."MV05 open" := "Data".Pot_MV05 < 98;
   "Inputs"."MV05 Close" := "Data".Pot_MV05 > 2;
   "Inputs"."MV06 Run_Opening" := "Open MV06";
   IF "Open MV06" AND "Clock100ms" AND ("Data".Pot_MV06 <= 100) THEN
       "Data".Pot_MV06 := "Data".Pot_MV06 + 1;
   END_IF;
   "Inputs"."MV06 Run_Closing" := "Close MV06";
   IF "Close MV06" AND "Clock100ms" AND ("Data".Pot_MV06 >= 0) THEN
       "Data".Pot_MV06 := "Data".Pot_MV06 - 1;
   END_IF;
   "Inputs".MV06_Open := "Data".Pot_MV06 >= 98;
   "Inputs"."MV06 Close" := "Data".Pot_MV06 <= 2;
END_REGION

REGION Network 6: Motors simulated
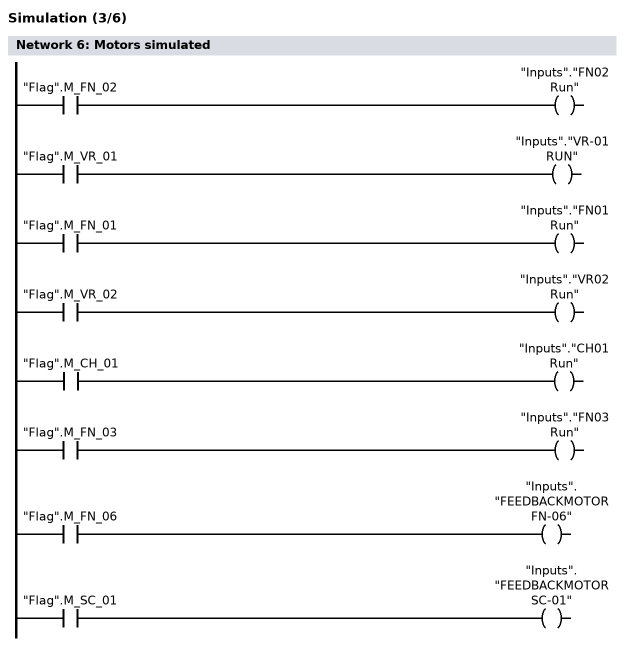
   RUNG wire#powerrail
      Contact( "Flag".M_FN_02 )
      Coil( "Inputs"."FN02 Run" )
   END_RUNG
   RUNG wire#powerrail
      Contact( "Flag".M_VR_01 )
      Coil( "Inputs"."VR-01 RUN" )
   END_RUNG
   RUNG wire#powerrail
      Contact( "Flag".M_FN_01 )
      Coil( "Inputs"."FN01 Run" )
   END_RUNG
   RUNG wire#powerrail
      Contact( "Flag".M_VR_02 )
      Coil( "Inputs"."VR02 Run" )
   END_RUNG
   RUNG wire#powerrail
      Contact( "Flag".M_CH_01 )
      Coil( "Inputs"."CH01 Run" )
   END_RUNG
   RUNG wire#powerrail
      Contact( "Flag".M_FN_03 )
      Coil( "Inputs"."FN03 Run" )
   END_RUNG
   RUNG wire#powerrail
      Contact( "Flag".M_FN_06 )
      Coil( "Inputs"."FEEDBACKMOTOR FN-06" )
   END_RUNG
   RUNG wire#powerrail
      Contact( "Flag".M_SC_01 )
      Coil( "Inputs"."FEEDBACKMOTOR SC-01" )
   END_RUNG
   // the same network as SCL:
   "Inputs"."FN02 Run" := "Flag".M_FN_02;
   "Inputs"."VR-01 RUN" := "Flag".M_VR_01;
   "Inputs"."FN01 Run" := "Flag".M_FN_01;
   "Inputs"."VR02 Run" := "Flag".M_VR_02;
   "Inputs"."CH01 Run" := "Flag".M_CH_01;
   "Inputs"."FN03 Run" := "Flag".M_FN_03;
   "Inputs"."FEEDBACKMOTOR FN-06" := "Flag".M_FN_06;
   "Inputs"."FEEDBACKMOTOR SC-01" := "Flag".M_SC_01;
END_REGION

REGION Network 7: Motors simulated
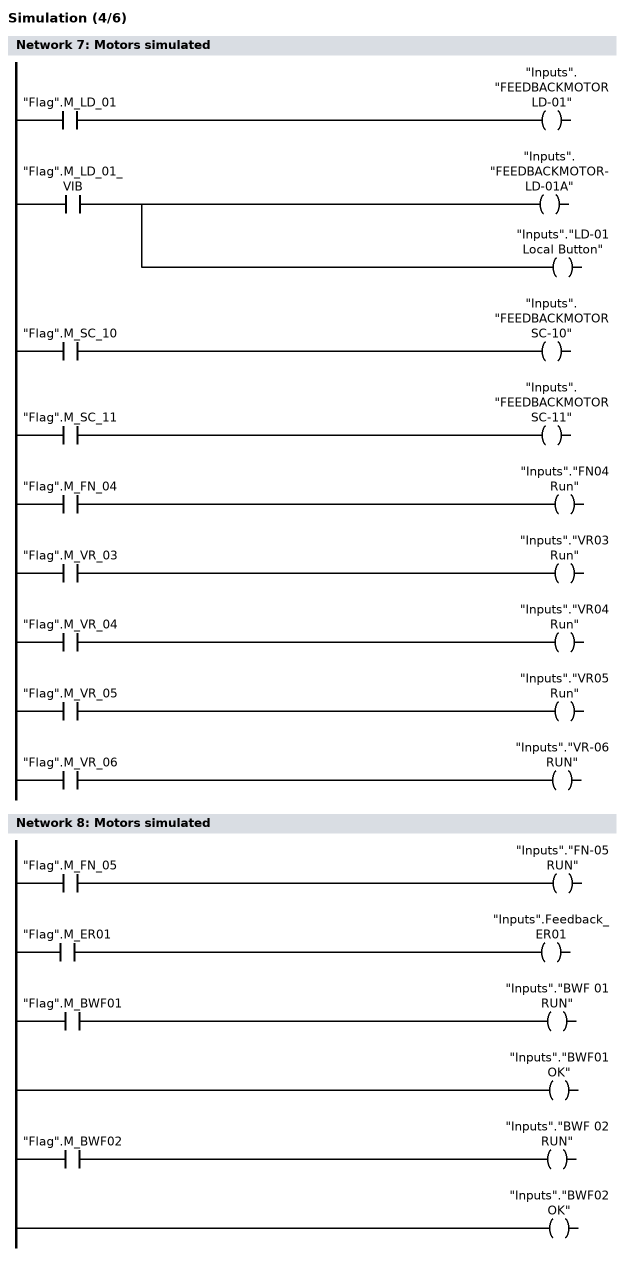
   RUNG wire#powerrail
      Contact( "Flag".M_LD_01 )
      Coil( "Inputs"."FEEDBACKMOTOR LD-01" )
   END_RUNG
   RUNG wire#powerrail
      Contact( "Flag".M_LD_01_VIB )
      wire#w1
      Coil( "Inputs"."FEEDBACKMOTOR-LD-01A" )
   END_RUNG
   RUNG wire#w1
      Coil( "Inputs"."LD-01 Local Button" )
   END_RUNG
   RUNG wire#powerrail
      Contact( "Flag".M_SC_10 )
      Coil( "Inputs"."FEEDBACKMOTOR SC-10" )
   END_RUNG
   RUNG wire#powerrail
      Contact( "Flag".M_SC_11 )
      Coil( "Inputs"."FEEDBACKMOTOR SC-11" )
   END_RUNG
   RUNG wire#powerrail
      Contact( "Flag".M_FN_04 )
      Coil( "Inputs"."FN04 Run" )
   END_RUNG
   RUNG wire#powerrail
      Contact( "Flag".M_VR_03 )
      Coil( "Inputs"."VR03 Run" )
   END_RUNG
   RUNG wire#powerrail
      Contact( "Flag".M_VR_04 )
      Coil( "Inputs"."VR04 Run" )
   END_RUNG
   RUNG wire#powerrail
      Contact( "Flag".M_VR_05 )
      Coil( "Inputs"."VR05 Run" )
   END_RUNG
   RUNG wire#powerrail
      Contact( "Flag".M_VR_06 )
      Coil( "Inputs"."VR-06 RUN" )
   END_RUNG
   // the same network as SCL:
   "Inputs"."FEEDBACKMOTOR LD-01" := "Flag".M_LD_01;
   "Inputs"."FEEDBACKMOTOR-LD-01A" := "Flag".M_LD_01_VIB;
   "Inputs"."LD-01 Local Button" := "Flag".M_LD_01_VIB;
   "Inputs"."FEEDBACKMOTOR SC-10" := "Flag".M_SC_10;
   "Inputs"."FEEDBACKMOTOR SC-11" := "Flag".M_SC_11;
   "Inputs"."FN04 Run" := "Flag".M_FN_04;
   "Inputs"."VR03 Run" := "Flag".M_VR_03;
   "Inputs"."VR04 Run" := "Flag".M_VR_04;
   "Inputs"."VR05 Run" := "Flag".M_VR_05;
   "Inputs"."VR-06 RUN" := "Flag".M_VR_06;
END_REGION

REGION Network 8: Motors simulated
   RUNG wire#powerrail
      Contact( "Flag".M_FN_05 )
      Coil( "Inputs"."FN-05 RUN" )
   END_RUNG
   RUNG wire#powerrail
      Contact( "Flag".M_ER01 )
      Coil( "Inputs".Feedback_ER01 )
   END_RUNG
   RUNG wire#powerrail
      Contact( "Flag".M_BWF01 )
      Coil( "Inputs"."BWF 01 RUN" )
   END_RUNG
   RUNG wire#powerrail
      Coil( "Inputs"."BWF01 OK" )
   END_RUNG
   RUNG wire#powerrail
      Contact( "Flag".M_BWF02 )
      Coil( "Inputs"."BWF 02 RUN" )
   END_RUNG
   RUNG wire#powerrail
      Coil( "Inputs"."BWF02 OK" )
   END_RUNG
   // the same network as SCL:
   "Inputs"."FN-05 RUN" := "Flag".M_FN_05;
   "Inputs".Feedback_ER01 := "Flag".M_ER01;
   "Inputs"."BWF 01 RUN" := "Flag".M_BWF01;
   "Inputs"."BWF01 OK" := TRUE;
   "Inputs"."BWF 02 RUN" := "Flag".M_BWF02;
   "Inputs"."BWF02 OK" := TRUE;
END_REGION

REGION Network 9: pv03
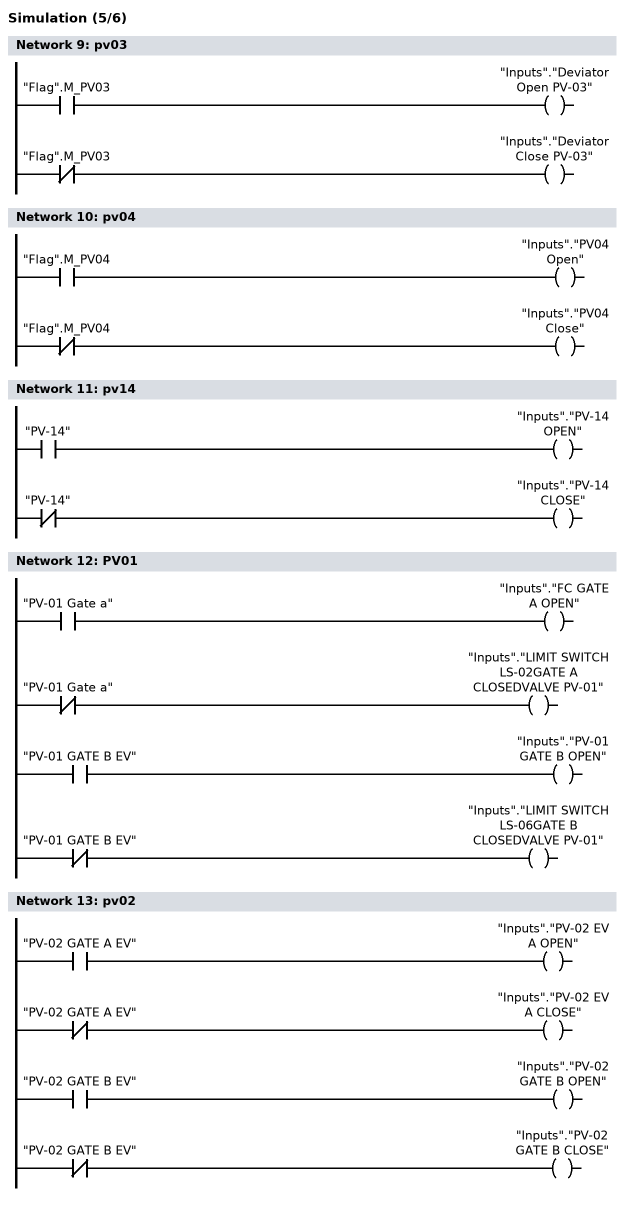
   RUNG wire#powerrail
      Contact( "Flag".M_PV03 )
      Coil( "Inputs"."Deviator Open PV-03" )
   END_RUNG
   RUNG wire#powerrail
      I_Contact( "Flag".M_PV03 )
      Coil( "Inputs"."Deviator Close PV-03" )
   END_RUNG
   // the same network as SCL:
   "Inputs"."Deviator Open PV-03" := "Flag".M_PV03;
   "Inputs"."Deviator Close PV-03" := NOT "Flag".M_PV03;
END_REGION

REGION Network 10: pv04
   RUNG wire#powerrail
      Contact( "Flag".M_PV04 )
      Coil( "Inputs"."PV04 Open" )
   END_RUNG
   RUNG wire#powerrail
      I_Contact( "Flag".M_PV04 )
      Coil( "Inputs"."PV04 Close" )
   END_RUNG
   // the same network as SCL:
   "Inputs"."PV04 Open" := "Flag".M_PV04;
   "Inputs"."PV04 Close" := NOT "Flag".M_PV04;
END_REGION

REGION Network 11: pv14
   RUNG wire#powerrail
      Contact( "PV-14" )
      Coil( "Inputs"."PV-14 OPEN" )
   END_RUNG
   RUNG wire#powerrail
      I_Contact( "PV-14" )
      Coil( "Inputs"."PV-14 CLOSE" )
   END_RUNG
   // the same network as SCL:
   "Inputs"."PV-14 OPEN" := "PV-14";
   "Inputs"."PV-14 CLOSE" := NOT "PV-14";
END_REGION

REGION Network 12: PV01
   RUNG wire#powerrail
      Contact( "PV-01 Gate a" )
      Coil( "Inputs"."FC GATE A OPEN" )
   END_RUNG
   RUNG wire#powerrail
      I_Contact( "PV-01 Gate a" )
      Coil( "Inputs"."LIMIT SWITCH LS-02GATE A CLOSEDVALVE PV-01" )
   END_RUNG
   RUNG wire#powerrail
      Contact( "PV-01 GATE B EV" )
      Coil( "Inputs"."PV-01 GATE B OPEN" )
   END_RUNG
   RUNG wire#powerrail
      I_Contact( "PV-01 GATE B EV" )
      Coil( "Inputs"."LIMIT SWITCH LS-06GATE B CLOSEDVALVE PV-01" )
   END_RUNG
   // the same network as SCL:
   "Inputs"."FC GATE A OPEN" := "PV-01 Gate a";
   "Inputs"."LIMIT SWITCH LS-02GATE A CLOSEDVALVE PV-01" := NOT "PV-01 Gate a";
   "Inputs"."PV-01 GATE B OPEN" := "PV-01 GATE B EV";
   "Inputs"."LIMIT SWITCH LS-06GATE B CLOSEDVALVE PV-01" := NOT "PV-01 GATE B EV";
END_REGION

REGION Network 13: pv02
   RUNG wire#powerrail
      Contact( "PV-02 GATE A EV" )
      Coil( "Inputs"."PV-02 EV A OPEN" )
   END_RUNG
   RUNG wire#powerrail
      I_Contact( "PV-02 GATE A EV" )
      Coil( "Inputs"."PV-02 EV A CLOSE" )
   END_RUNG
   RUNG wire#powerrail
      Contact( "PV-02 GATE B EV" )
      Coil( "Inputs"."PV-02 GATE B OPEN" )
   END_RUNG
   RUNG wire#powerrail
      I_Contact( "PV-02 GATE B EV" )
      Coil( "Inputs"."PV-02 GATE B CLOSE" )
   END_RUNG
   // the same network as SCL:
   "Inputs"."PV-02 EV A OPEN" := "PV-02 GATE A EV";
   "Inputs"."PV-02 EV A CLOSE" := NOT "PV-02 GATE A EV";
   "Inputs"."PV-02 GATE B OPEN" := "PV-02 GATE B EV";
   "Inputs"."PV-02 GATE B CLOSE" := NOT "PV-02 GATE B EV";
END_REGION

REGION Network 14
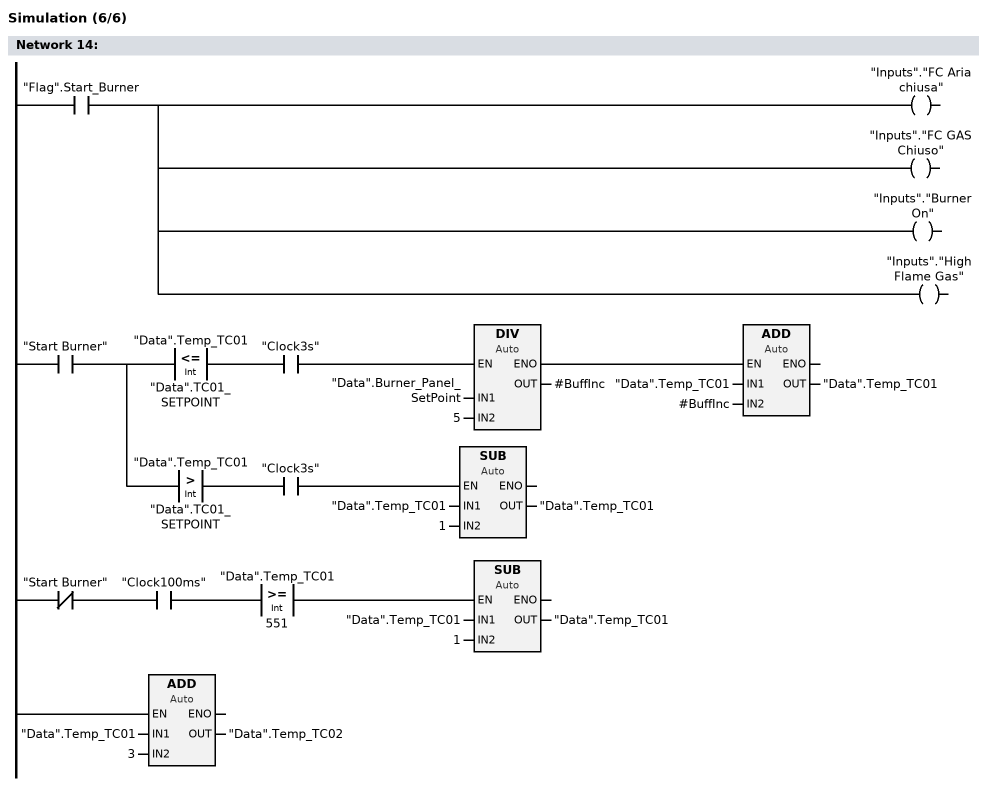
   RUNG wire#powerrail
      Contact( "Flag".Start_Burner )
      wire#w1
      Coil( "Inputs"."FC Aria chiusa" )
   END_RUNG
   RUNG wire#w1
      Coil( "Inputs"."FC GAS Chiuso" )
   END_RUNG
   RUNG wire#w1
      Coil( "Inputs"."Burner On" )
   END_RUNG
   RUNG wire#w1
      Coil( "Inputs"."High Flame Gas" )
   END_RUNG
   RUNG wire#powerrail
      Contact( "Start Burner" )
      wire#w2
      { S7_Templates := "SrcType := Int" } LE_Contact(in1 := "Data".Temp_TC01, in2 := "Data".TC01_SETPOINT)
      Contact( "Clock3s" )
      Div(in1 := "Data".Burner_Panel_SetPoint, in2 := 5, out => #BuffInc)
      Add(in1 := "Data".Temp_TC01, in2 := #BuffInc, out => "Data".Temp_TC01)
   END_RUNG
   RUNG wire#w2
      { S7_Templates := "SrcType := Int" } GT_Contact(in1 := "Data".Temp_TC01, in2 := "Data".TC01_SETPOINT)
      Contact( "Clock3s" )
      Sub(in1 := "Data".Temp_TC01, in2 := 1, out => "Data".Temp_TC01)
   END_RUNG
   RUNG wire#powerrail
      I_Contact( "Start Burner" )
      Contact( "Clock100ms" )
      { S7_Templates := "SrcType := Int" } GE_Contact(in1 := "Data".Temp_TC01, in2 := 551)
      Sub(in1 := "Data".Temp_TC01, in2 := 1, out => "Data".Temp_TC01)
   END_RUNG
   RUNG wire#powerrail
      Add(in1 := "Data".Temp_TC01, in2 := 3, out => "Data".Temp_TC02)
   END_RUNG
   // the same network as SCL:
   "Inputs"."FC Aria chiusa" := "Flag".Start_Burner;
   "Inputs"."FC GAS Chiuso" := "Flag".Start_Burner;
   "Inputs"."Burner On" := "Flag".Start_Burner;
   "Inputs"."High Flame Gas" := "Flag".Start_Burner;
   IF "Start Burner" AND ("Data".Temp_TC01 <= "Data".TC01_SETPOINT) AND "Clock3s" THEN
       #BuffInc := "Data".Burner_Panel_SetPoint / 5;
       "Data".Temp_TC01 := "Data".Temp_TC01 + #BuffInc;
   END_IF;
   IF "Start Burner" AND ("Data".Temp_TC01 > "Data".TC01_SETPOINT) AND "Clock3s" THEN
       "Data".Temp_TC01 := "Data".Temp_TC01 - 1;
   END_IF;
   IF NOT "Start Burner" AND "Clock100ms" AND ("Data".Temp_TC01 >= 551) THEN
       "Data".Temp_TC01 := "Data".Temp_TC01 - 1;
   END_IF;
   "Data".Temp_TC02 := "Data".Temp_TC01 + 3;
END_REGION
END_FUNCTION

FUNCTION "Allarm manager" : Void   // FC24, LAD
{ S7_Optimized_Access := 'FALSE' }
VERSION : 0.1
   VAR_TEMP   // added for the SCL form of the ladder/FBD networks
      _w1 : Bool;
      _w2 : Bool;
   END_VAR
BEGIN

REGION Network 1: MANAGEMENT ALARMS
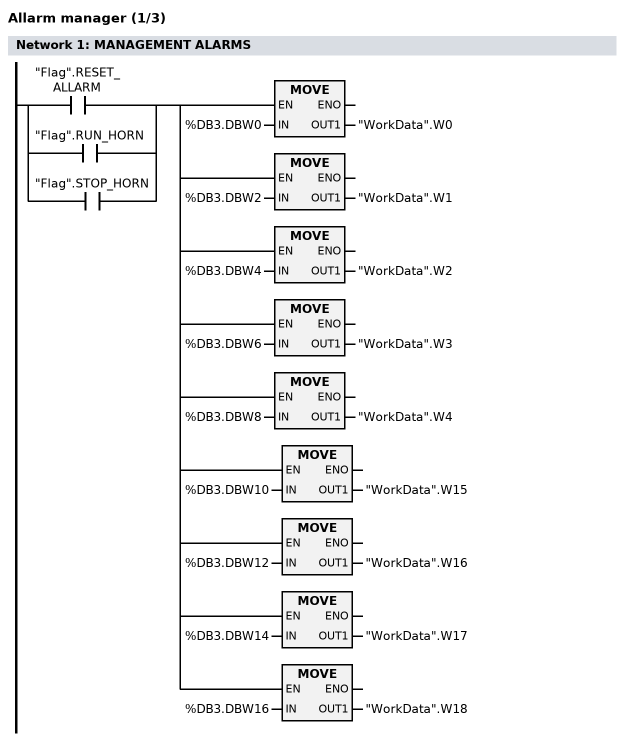
   RUNG wire#powerrail
      Contact( "Flag".RESET_ALLARM )
      wire#w1
      { S7_GenerateENO := "TRUE" } Move(in := %DB3.DBW0, out1 => "WorkData".W0)
   END_RUNG
   RUNG wire#powerrail
      Contact( "Flag".RUN_HORN )
   END_RUNG wire#w1
   RUNG wire#powerrail
      Contact( "Flag".STOP_HORN )
   END_RUNG wire#w1
   RUNG wire#w1
      { S7_GenerateENO := "TRUE" } Move(in := %DB3.DBW2, out1 => "WorkData".W1)
   END_RUNG
   RUNG wire#w1
      { S7_GenerateENO := "TRUE" } Move(in := %DB3.DBW4, out1 => "WorkData".W2)
   END_RUNG
   RUNG wire#w1
      { S7_GenerateENO := "TRUE" } Move(in := %DB3.DBW6, out1 => "WorkData".W3)
   END_RUNG
   RUNG wire#w1
      { S7_GenerateENO := "TRUE" } Move(in := %DB3.DBW8, out1 => "WorkData".W4)
   END_RUNG
   RUNG wire#w1
      { S7_GenerateENO := "TRUE" } Move(in := %DB3.DBW10, out1 => "WorkData".W15)
   END_RUNG
   RUNG wire#w1
      { S7_GenerateENO := "TRUE" } Move(in := %DB3.DBW12, out1 => "WorkData".W16)
   END_RUNG
   RUNG wire#w1
      { S7_GenerateENO := "TRUE" } Move(in := %DB3.DBW14, out1 => "WorkData".W17)
   END_RUNG
   RUNG wire#w1
      { S7_GenerateENO := "TRUE" } Move(in := %DB3.DBW16, out1 => "WorkData".W18)
   END_RUNG
   // the same network as SCL:
   IF "Flag".RESET_ALLARM OR "Flag".RUN_HORN OR "Flag".STOP_HORN THEN
       "WorkData".W0 := %DB3.DBW0;
       "WorkData".W1 := %DB3.DBW2;
       "WorkData".W2 := %DB3.DBW4;
       "WorkData".W3 := %DB3.DBW6;
       "WorkData".W4 := %DB3.DBW8;
       "WorkData".W15 := %DB3.DBW10;
       "WorkData".W16 := %DB3.DBW12;
       "WorkData".W17 := %DB3.DBW14;
       "WorkData".W18 := %DB3.DBW16;
   END_IF;
END_REGION

REGION Network 2: COM_W3 BIT11 (NEW_ALLARM)
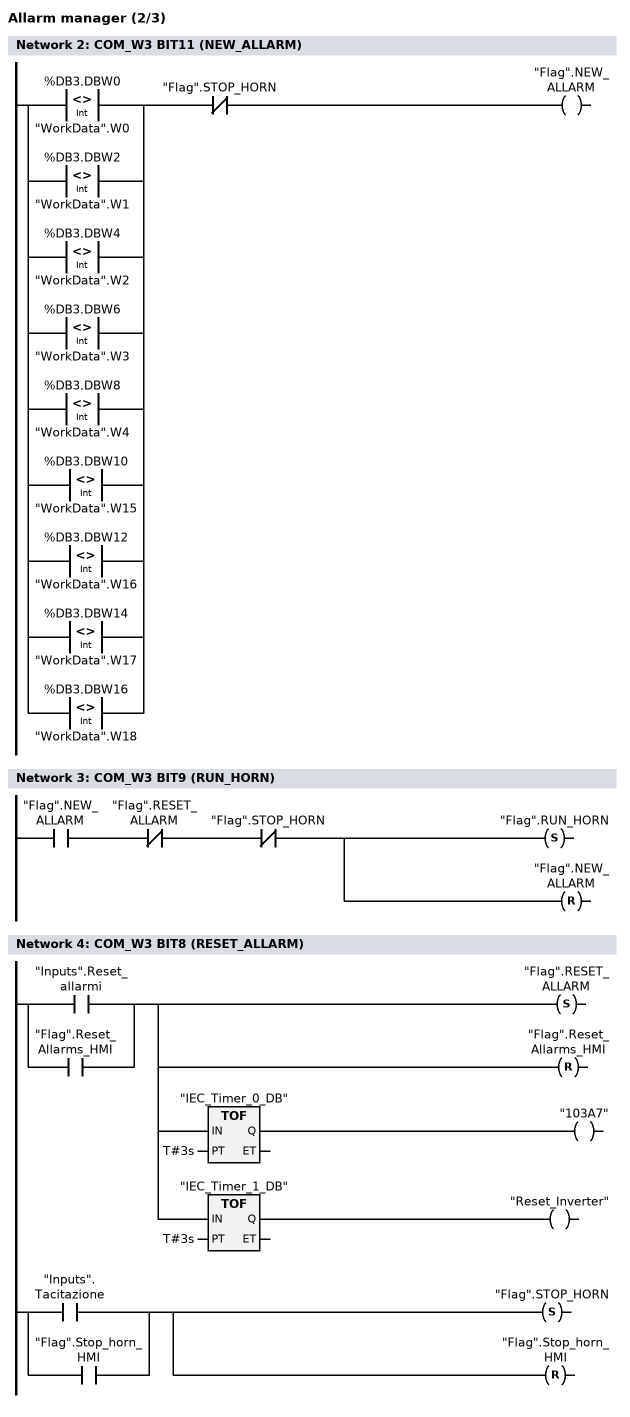
   RUNG wire#powerrail
      { S7_Templates := "SrcType := Int" } NE_Contact(in1 := %DB3.DBW0, in2 := "WorkData".W0)
      wire#w1
      I_Contact( "Flag".STOP_HORN )
      Coil( "Flag".NEW_ALLARM )
   END_RUNG
   RUNG wire#powerrail
      { S7_Templates := "SrcType := Int" } NE_Contact(in1 := %DB3.DBW2, in2 := "WorkData".W1)
   END_RUNG wire#w1
   RUNG wire#powerrail
      { S7_Templates := "SrcType := Int" } NE_Contact(in1 := %DB3.DBW4, in2 := "WorkData".W2)
   END_RUNG wire#w1
   RUNG wire#powerrail
      { S7_Templates := "SrcType := Int" } NE_Contact(in1 := %DB3.DBW6, in2 := "WorkData".W3)
   END_RUNG wire#w1
   RUNG wire#powerrail
      { S7_Templates := "SrcType := Int" } NE_Contact(in1 := %DB3.DBW8, in2 := "WorkData".W4)
   END_RUNG wire#w1
   RUNG wire#powerrail
      { S7_Templates := "SrcType := Int" } NE_Contact(in1 := %DB3.DBW10, in2 := "WorkData".W15)
   END_RUNG wire#w1
   RUNG wire#powerrail
      { S7_Templates := "SrcType := Int" } NE_Contact(in1 := %DB3.DBW12, in2 := "WorkData".W16)
   END_RUNG wire#w1
   RUNG wire#powerrail
      { S7_Templates := "SrcType := Int" } NE_Contact(in1 := %DB3.DBW14, in2 := "WorkData".W17)
   END_RUNG wire#w1
   RUNG wire#powerrail
      { S7_Templates := "SrcType := Int" } NE_Contact(in1 := %DB3.DBW16, in2 := "WorkData".W18)
   END_RUNG wire#w1
   // the same network as SCL:
   "Flag".NEW_ALLARM := ((%DB3.DBW0 <> "WorkData".W0) OR (%DB3.DBW2 <> "WorkData".W1) OR (%DB3.DBW4 <> "WorkData".W2) OR (%DB3.DBW6 <> "WorkData".W3) OR (%DB3.DBW8 <> "WorkData".W4) OR (%DB3.DBW10 <> "WorkData".W15) OR (%DB3.DBW12 <> "WorkData".W16) OR (%DB3.DBW14 <> "WorkData".W17) OR (%DB3.DBW16 <> "WorkData".W18)) AND NOT "Flag".STOP_HORN;
END_REGION

REGION Network 3: COM_W3 BIT9 (RUN_HORN)
   RUNG wire#powerrail
      Contact( "Flag".NEW_ALLARM )
      I_Contact( "Flag".RESET_ALLARM )
      I_Contact( "Flag".STOP_HORN )
      wire#w1
      S_Coil( "Flag".RUN_HORN )
   END_RUNG
   RUNG wire#w1
      R_Coil( "Flag".NEW_ALLARM )
   END_RUNG
   // the same network as SCL:
   IF "Flag".NEW_ALLARM AND NOT "Flag".RESET_ALLARM AND NOT "Flag".STOP_HORN THEN
       "Flag".RUN_HORN := TRUE;
       "Flag".NEW_ALLARM := FALSE;
   END_IF;
END_REGION

REGION Network 4: COM_W3 BIT8 (RESET_ALLARM)
   #_w1 := "Inputs".Reset_allarmi OR "Flag".Reset_Allarms_HMI;
   IF #_w1 THEN
       "Flag".RESET_ALLARM := TRUE;
       "Flag".Reset_Allarms_HMI := FALSE;
   END_IF;
   "IEC_Timer_0_DB".TOF(IN := #_w1, PT := T#3s);
   "103A7" := "IEC_Timer_0_DB".Q;
   "IEC_Timer_1_DB".TOF(IN := #_w1, PT := T#3s);
   "Reset_Inverter" := "IEC_Timer_1_DB".Q;
   IF "Inputs".Tacitazione OR "Flag".Stop_horn_HMI THEN
       "Flag".STOP_HORN := TRUE;
       "Flag".Stop_horn_HMI := FALSE;
   END_IF;
END_REGION

REGION Network 5: COM_W3 BIT8 (RESET_ALLARM)
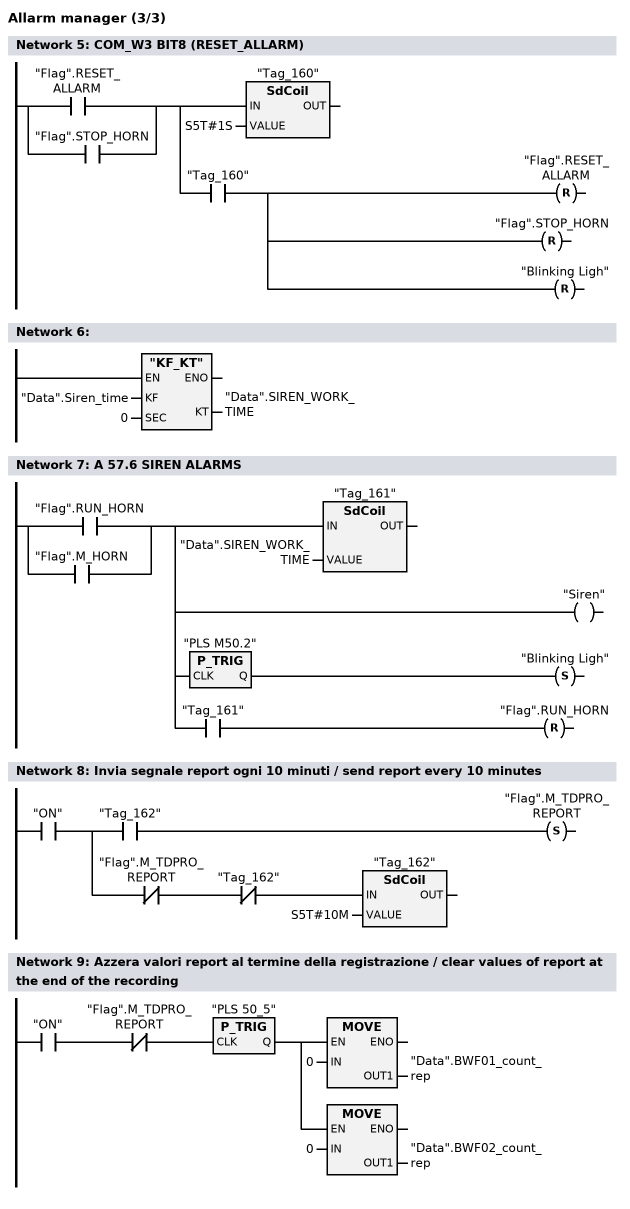
   // no SCL statement known for SdCoil: written as a call
   #_w1 := "Flag".RESET_ALLARM OR "Flag".STOP_HORN;
   SdCoil(in := #_w1, value := S5T#1S, operand := "Tag_160");
   IF #_w1 AND "Tag_160" THEN
       "Flag".RESET_ALLARM := FALSE;
       "Flag".STOP_HORN := FALSE;
       "Blinking Ligh" := FALSE;
   END_IF;
END_REGION

REGION Network 6
   RUNG wire#powerrail
      "KF_KT"(KF := "Data".Siren_time, SEC := 0, KT => "Data".SIREN_WORK_TIME)
   END_RUNG
   // the same network as SCL:
   "KF_KT"(KF := "Data".Siren_time, SEC := 0, KT => "Data".SIREN_WORK_TIME);
END_REGION

REGION Network 7: A 57.6 SIREN ALARMS
   // no SCL statement known for SdCoil: written as a call
   #_w1 := "Flag".RUN_HORN OR "Flag".M_HORN;
   SdCoil(in := #_w1, value := "Data".SIREN_WORK_TIME, operand := "Tag_161");
   "Siren" := #_w1;
   #_w2 := #_w1 AND NOT "PLS M50.2";   // rising edge
   "PLS M50.2" := #_w1;
   IF #_w2 THEN "Blinking Ligh" := TRUE; END_IF;
   IF #_w1 AND "Tag_161" THEN "Flag".RUN_HORN := FALSE; END_IF;
END_REGION

REGION Network 8: Invia segnale report ogni 10 minuti / send report every 10 minutes
   // no SCL statement known for SdCoil: written as a call
   IF "ON" AND "Tag_162" THEN "Flag".M_TDPRO_REPORT := TRUE; END_IF;
   SdCoil(in := "ON" AND NOT "Flag".M_TDPRO_REPORT AND NOT "Tag_162", value := S5T#10M, operand := "Tag_162");
END_REGION

REGION Network 9: Azzera valori report al termine della registrazione / clear values of report at the end of the recording
   RUNG wire#powerrail
      Contact( "ON" )
      I_Contact( "Flag".M_TDPRO_REPORT )
      P_Trig( "PLS 50_5" )
      wire#w1
      { S7_GenerateENO := "TRUE" } Move(in := 0, out1 => "Data".BWF01_count_rep)
   END_RUNG
   RUNG wire#w1
      { S7_GenerateENO := "TRUE" } Move(in := 0, out1 => "Data".BWF02_count_rep)
   END_RUNG
   // the same network as SCL:
   #_w1 := "ON" AND NOT "Flag".M_TDPRO_REPORT;
   #_w2 := #_w1 AND NOT "PLS 50_5";   // rising edge
   "PLS 50_5" := #_w1;
   IF #_w2 THEN
       "Data".BWF01_count_rep := 0;
       "Data".BWF02_count_rep := 0;
   END_IF;
END_REGION
END_FUNCTION

FUNCTION "Auto start motors" : Void   // FC30, LAD
TITLE = Questa FC viene richiamata ogni 1sec / This FC is recalled every 1ms
{ S7_Optimized_Access := 'FALSE' }
VERSION : 0.1
   VAR_TEMP
      Prod_h_bwf01 : Real;
      Prod_h_bwf02 : Real;
      Prod_h : Real;
      Prod_s_bwf01 : Real;
      Prod_s_bwf02 : Real;
   END_VAR
   VAR_TEMP   // added for the SCL form of the ladder/FBD networks
      _w1 : Bool;
      _w2 : Bool;
      _w3 : Bool;
   END_VAR
BEGIN

REGION Network 1: Incrementa conteggio secondi / Increment seconds count
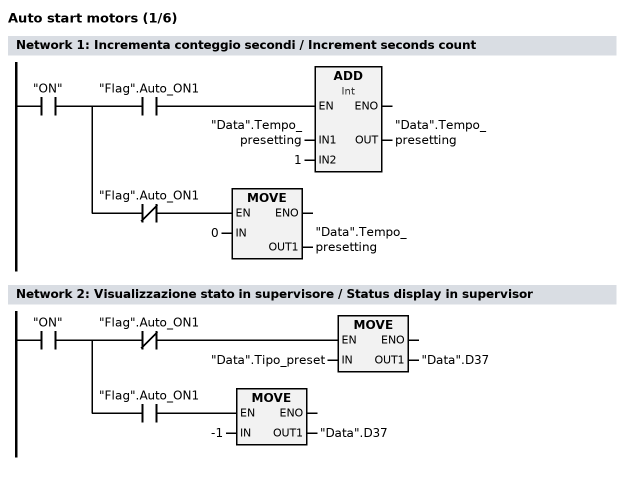
   RUNG wire#powerrail
      Contact( "ON" )
      wire#w1
      Contact( "Flag".Auto_ON1 )
      { S7_Templates := "SrcType := Int"; S7_GenerateENO := "TRUE" } Add(in1 := "Data".Tempo_presetting, in2 := 1, out => "Data".Tempo_presetting)
   END_RUNG
   RUNG wire#w1
      I_Contact( "Flag".Auto_ON1 )
      { S7_GenerateENO := "TRUE" } Move(in := 0, out1 => "Data".Tempo_presetting)
   END_RUNG
   // the same network as SCL:
   IF "ON" AND "Flag".Auto_ON1 THEN "Data".Tempo_presetting := "Data".Tempo_presetting + 1; END_IF;
   IF "ON" AND NOT "Flag".Auto_ON1 THEN "Data".Tempo_presetting := 0; END_IF;
END_REGION

REGION Network 2: Visualizzazione stato in supervisore / Status display in supervisor
   RUNG wire#powerrail
      Contact( "ON" )
      wire#w1
      I_Contact( "Flag".Auto_ON1 )
      { S7_GenerateENO := "TRUE" } Move(in := "Data".Tipo_preset, out1 => "Data".D37)
   END_RUNG
   RUNG wire#w1
      Contact( "Flag".Auto_ON1 )
      { S7_GenerateENO := "TRUE" } Move(in := -1, out1 => "Data".D37)
   END_RUNG
   // the same network as SCL:
   IF "ON" AND NOT "Flag".Auto_ON1 THEN "Data".D37 := "Data".Tipo_preset; END_IF;
   IF "ON" AND "Flag".Auto_ON1 THEN "Data".D37 := -1; END_IF;
END_REGION

REGION Network 3: Sequenza di PRERICALDO O STANDBY / PREHEATING
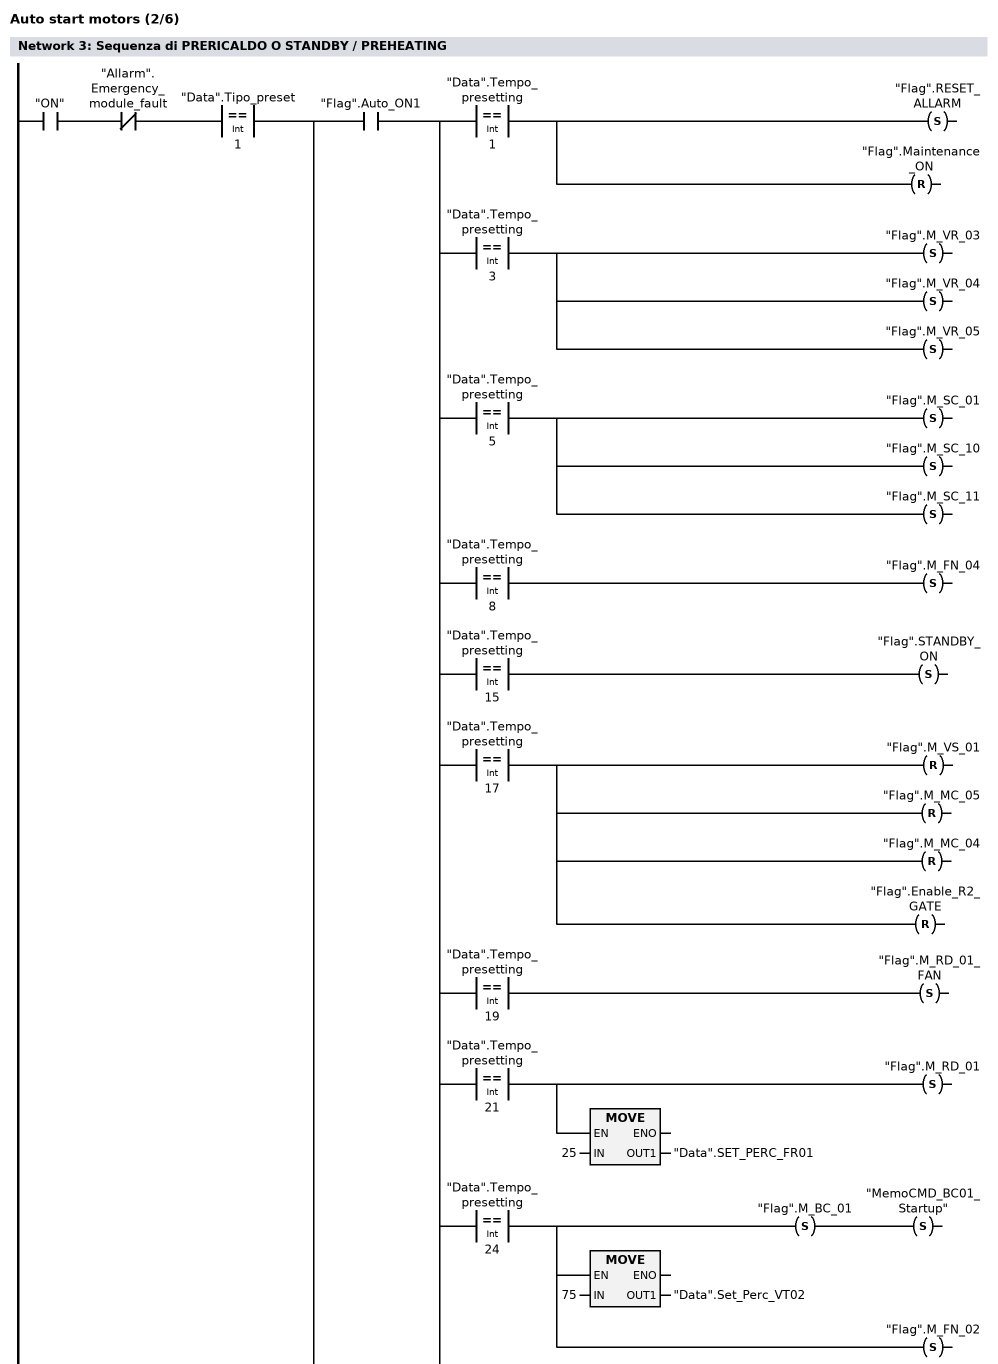
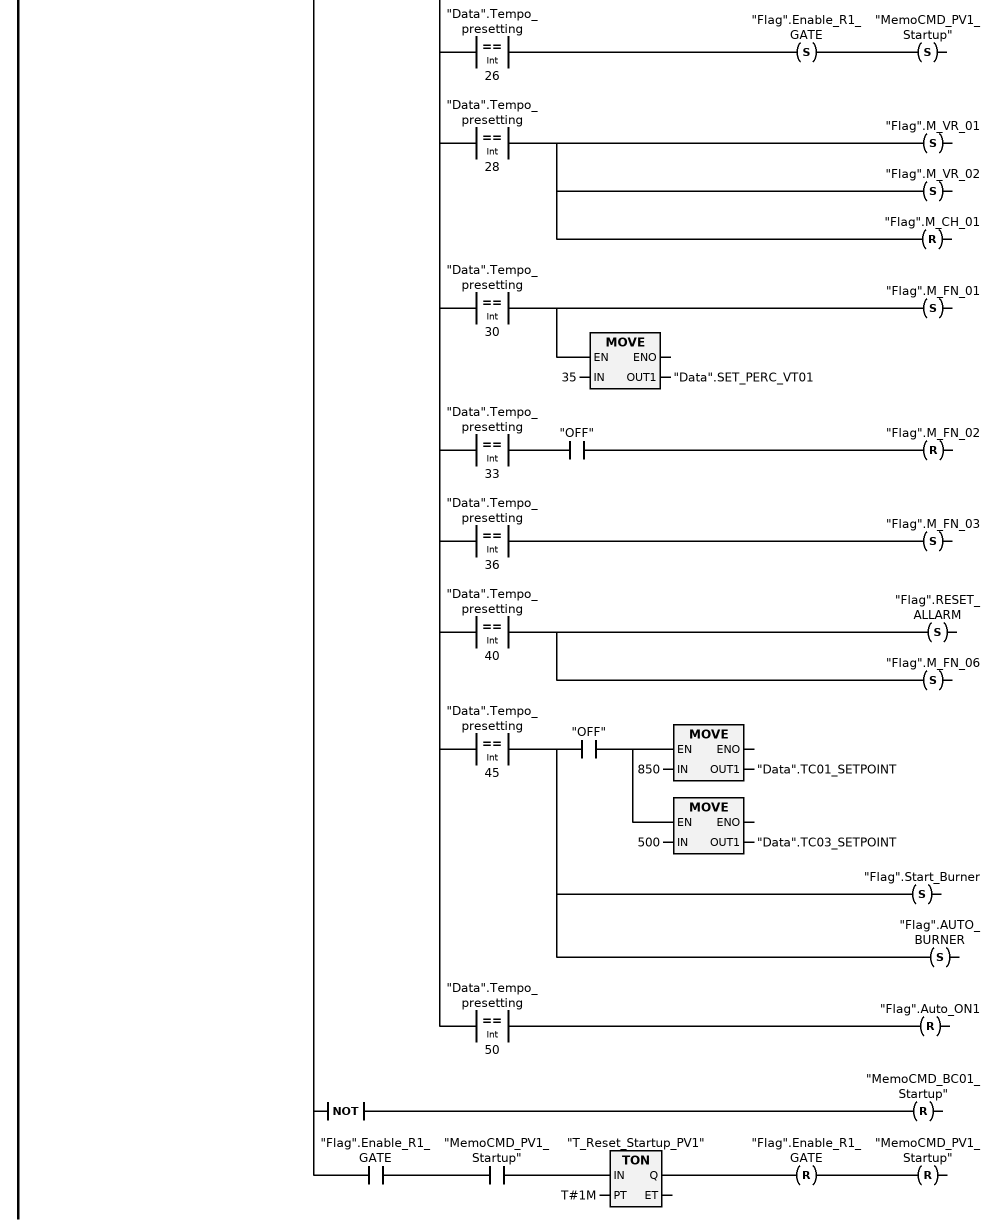
   #_w1 := "ON" AND NOT "Allarm".Emergency_module_fault AND ("Data".Tipo_preset = 1);
   #_w2 := #_w1 AND "Flag".Auto_ON1;
   IF #_w2 AND ("Data".Tempo_presetting = 1) THEN
       "Flag".RESET_ALLARM := TRUE;
       "Flag".Maintenance_ON := FALSE;
   END_IF;
   IF #_w2 AND ("Data".Tempo_presetting = 3) THEN
       "Flag".M_VR_03 := TRUE;
       "Flag".M_VR_04 := TRUE;
       "Flag".M_VR_05 := TRUE;
   END_IF;
   IF #_w2 AND ("Data".Tempo_presetting = 5) THEN
       "Flag".M_SC_01 := TRUE;
       "Flag".M_SC_10 := TRUE;
       "Flag".M_SC_11 := TRUE;
   END_IF;
   IF #_w2 AND ("Data".Tempo_presetting = 8) THEN "Flag".M_FN_04 := TRUE; END_IF;
   IF #_w2 AND ("Data".Tempo_presetting = 15) THEN "Flag".STANDBY_ON := TRUE; END_IF;
   IF #_w2 AND ("Data".Tempo_presetting = 17) THEN
       "Flag".M_VS_01 := FALSE;
       "Flag".M_MC_05 := FALSE;
       "Flag".M_MC_04 := FALSE;
       "Flag".Enable_R2_GATE := FALSE;
   END_IF;
   IF #_w2 AND ("Data".Tempo_presetting = 19) THEN "Flag".M_RD_01_FAN := TRUE; END_IF;
   IF #_w2 AND ("Data".Tempo_presetting = 21) THEN
       "Flag".M_RD_01 := TRUE;
       "Data".SET_PERC_FR01 := 25;
   END_IF;
   IF #_w2 AND ("Data".Tempo_presetting = 24) THEN
       "Flag".M_BC_01 := TRUE;
       "MemoCMD_BC01_Startup" := TRUE;
       "Data".Set_Perc_VT02 := 75;
       "Flag".M_FN_02 := TRUE;
   END_IF;
   IF #_w2 AND ("Data".Tempo_presetting = 26) THEN
       "Flag".Enable_R1_GATE := TRUE;
       "MemoCMD_PV1_Startup" := TRUE;
   END_IF;
   IF #_w2 AND ("Data".Tempo_presetting = 28) THEN
       "Flag".M_VR_01 := TRUE;
       "Flag".M_VR_02 := TRUE;
       "Flag".M_CH_01 := FALSE;
   END_IF;
   IF #_w2 AND ("Data".Tempo_presetting = 30) THEN
       "Flag".M_FN_01 := TRUE;
       "Data".SET_PERC_VT01 := 35;
   END_IF;
   IF #_w2 AND ("Data".Tempo_presetting = 33) AND "OFF" THEN "Flag".M_FN_02 := FALSE; END_IF;
   IF #_w2 AND ("Data".Tempo_presetting = 36) THEN "Flag".M_FN_03 := TRUE; END_IF;
   IF #_w2 AND ("Data".Tempo_presetting = 40) THEN
       "Flag".RESET_ALLARM := TRUE;
       "Flag".M_FN_06 := TRUE;
   END_IF;
   #_w3 := #_w2 AND ("Data".Tempo_presetting = 45);
   IF #_w3 AND "OFF" THEN
       "Data".TC01_SETPOINT := 850;
       "Data".TC03_SETPOINT := 500;
   END_IF;
   IF #_w3 THEN
       "Flag".Start_Burner := TRUE;
       "Flag".AUTO_BURNER := TRUE;
   END_IF;
   IF #_w2 AND ("Data".Tempo_presetting = 50) THEN "Flag".Auto_ON1 := FALSE; END_IF;
   IF NOT #_w1 THEN "MemoCMD_BC01_Startup" := FALSE; END_IF;
   "T_Reset_Startup_PV1".TON(IN := #_w1 AND "Flag".Enable_R1_GATE AND "MemoCMD_PV1_Startup", PT := T#1M);
   IF "T_Reset_Startup_PV1".Q THEN
       "Flag".Enable_R1_GATE := FALSE;
       "MemoCMD_PV1_Startup" := FALSE;
   END_IF;
END_REGION

REGION Network 4: Sequenza di START GENERICA / Production
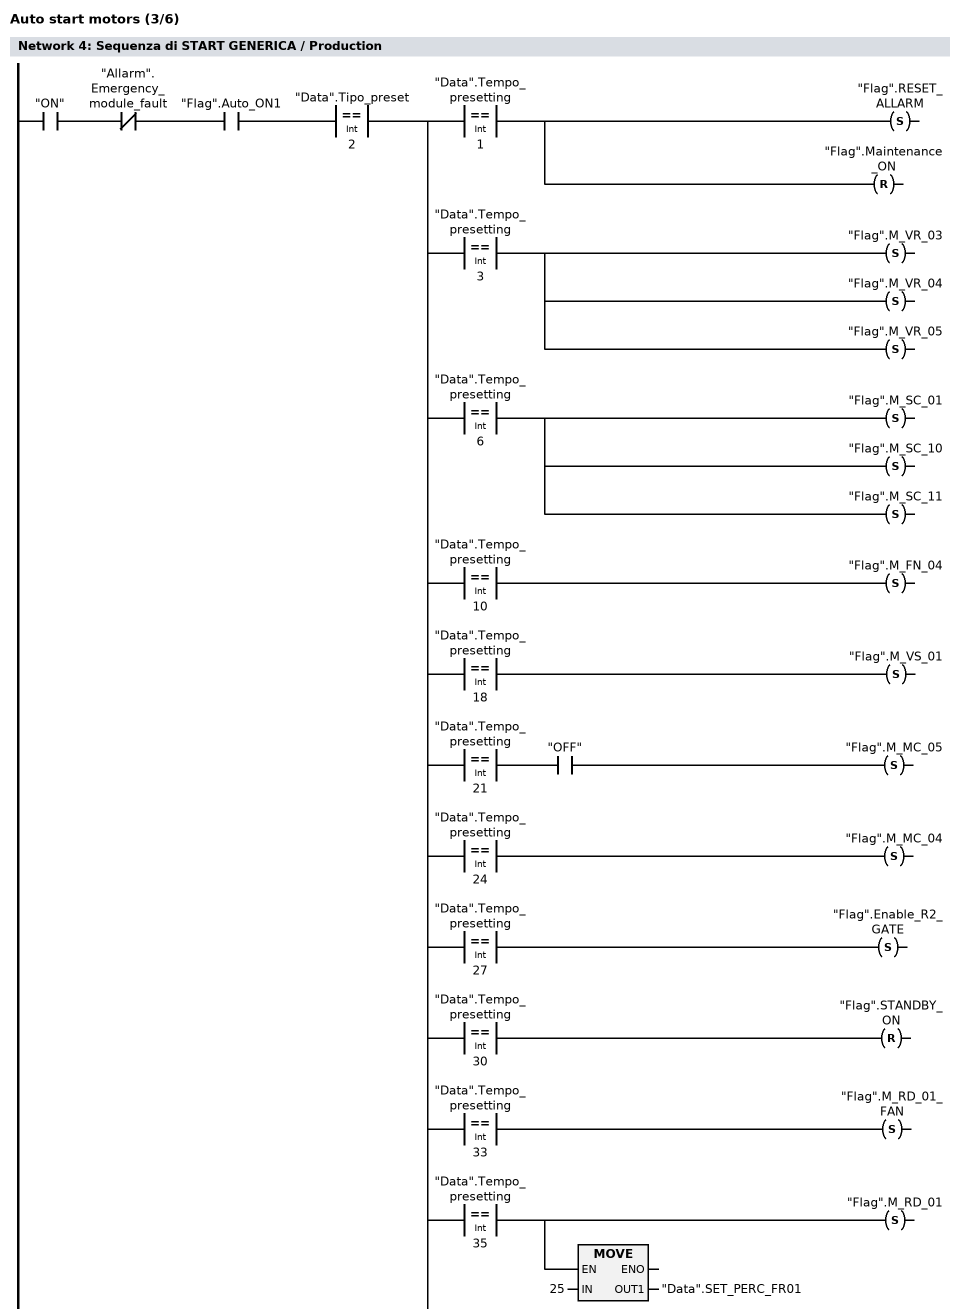
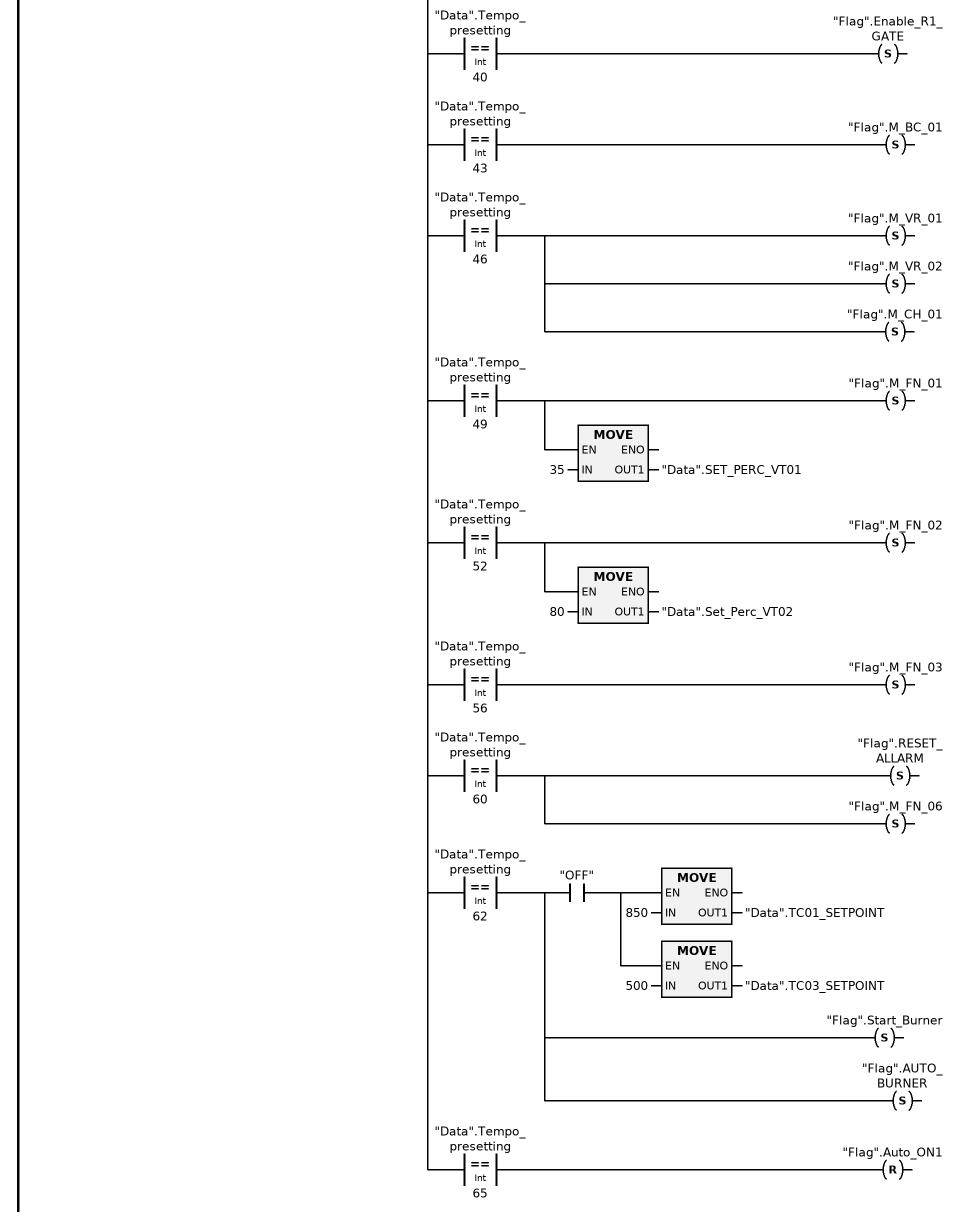
   RUNG wire#powerrail
      Contact( "ON" )
      I_Contact( "Allarm".Emergency_module_fault )
      Contact( "Flag".Auto_ON1 )
      { S7_Templates := "SrcType := Int" } EQ_Contact(in1 := "Data".Tipo_preset, in2 := 2)
      wire#w1
      { S7_Templates := "SrcType := Int" } EQ_Contact(in1 := "Data".Tempo_presetting, in2 := 1)
      wire#w2
      S_Coil( "Flag".RESET_ALLARM )
   END_RUNG
   RUNG wire#w2
      R_Coil( "Flag".Maintenance_ON )
   END_RUNG
   RUNG wire#w1
      { S7_Templates := "SrcType := Int" } EQ_Contact(in1 := "Data".Tempo_presetting, in2 := 3)
      wire#w3
      S_Coil( "Flag".M_VR_03 )
   END_RUNG
   RUNG wire#w3
      S_Coil( "Flag".M_VR_04 )
   END_RUNG
   RUNG wire#w3
      S_Coil( "Flag".M_VR_05 )
   END_RUNG
   RUNG wire#w1
      { S7_Templates := "SrcType := Int" } EQ_Contact(in1 := "Data".Tempo_presetting, in2 := 6)
      wire#w4
      S_Coil( "Flag".M_SC_01 )
   END_RUNG
   RUNG wire#w4
      S_Coil( "Flag".M_SC_10 )
   END_RUNG
   RUNG wire#w4
      S_Coil( "Flag".M_SC_11 )
   END_RUNG
   RUNG wire#w1
      { S7_Templates := "SrcType := Int" } EQ_Contact(in1 := "Data".Tempo_presetting, in2 := 10)
      S_Coil( "Flag".M_FN_04 )
   END_RUNG
   RUNG wire#w1
      { S7_Templates := "SrcType := Int" } EQ_Contact(in1 := "Data".Tempo_presetting, in2 := 18)
      S_Coil( "Flag".M_VS_01 )
   END_RUNG
   RUNG wire#w1
      { S7_Templates := "SrcType := Int" } EQ_Contact(in1 := "Data".Tempo_presetting, in2 := 21)
      Contact( "OFF" )
      S_Coil( "Flag".M_MC_05 )
   END_RUNG
   RUNG wire#w1
      { S7_Templates := "SrcType := Int" } EQ_Contact(in1 := "Data".Tempo_presetting, in2 := 24)
      S_Coil( "Flag".M_MC_04 )
   END_RUNG
   RUNG wire#w1
      { S7_Templates := "SrcType := Int" } EQ_Contact(in1 := "Data".Tempo_presetting, in2 := 27)
      S_Coil( "Flag".Enable_R2_GATE )
   END_RUNG
   RUNG wire#w1
      { S7_Templates := "SrcType := Int" } EQ_Contact(in1 := "Data".Tempo_presetting, in2 := 30)
      R_Coil( "Flag".STANDBY_ON )
   END_RUNG
   RUNG wire#w1
      { S7_Templates := "SrcType := Int" } EQ_Contact(in1 := "Data".Tempo_presetting, in2 := 33)
      S_Coil( "Flag".M_RD_01_FAN )
   END_RUNG
   RUNG wire#w1
      { S7_Templates := "SrcType := Int" } EQ_Contact(in1 := "Data".Tempo_presetting, in2 := 35)
      wire#w5
      S_Coil( "Flag".M_RD_01 )
   END_RUNG
   RUNG wire#w5
      { S7_GenerateENO := "TRUE" } Move(in := 25, out1 => "Data".SET_PERC_FR01)
   END_RUNG
   RUNG wire#w1
      { S7_Templates := "SrcType := Int" } EQ_Contact(in1 := "Data".Tempo_presetting, in2 := 40)
      S_Coil( "Flag".Enable_R1_GATE )
   END_RUNG
   RUNG wire#w1
      { S7_Templates := "SrcType := Int" } EQ_Contact(in1 := "Data".Tempo_presetting, in2 := 43)
      S_Coil( "Flag".M_BC_01 )
   END_RUNG
   RUNG wire#w1
      { S7_Templates := "SrcType := Int" } EQ_Contact(in1 := "Data".Tempo_presetting, in2 := 46)
      wire#w6
      S_Coil( "Flag".M_VR_01 )
   END_RUNG
   RUNG wire#w6
      S_Coil( "Flag".M_VR_02 )
   END_RUNG
   RUNG wire#w6
      S_Coil( "Flag".M_CH_01 )
   END_RUNG
   RUNG wire#w1
      { S7_Templates := "SrcType := Int" } EQ_Contact(in1 := "Data".Tempo_presetting, in2 := 49)
      wire#w7
      S_Coil( "Flag".M_FN_01 )
   END_RUNG
   RUNG wire#w7
      { S7_GenerateENO := "TRUE" } Move(in := 35, out1 => "Data".SET_PERC_VT01)
   END_RUNG
   RUNG wire#w1
      { S7_Templates := "SrcType := Int" } EQ_Contact(in1 := "Data".Tempo_presetting, in2 := 52)
      wire#w8
      S_Coil( "Flag".M_FN_02 )
   END_RUNG
   RUNG wire#w8
      { S7_GenerateENO := "TRUE" } Move(in := 80, out1 => "Data".Set_Perc_VT02)
   END_RUNG
   RUNG wire#w1
      { S7_Templates := "SrcType := Int" } EQ_Contact(in1 := "Data".Tempo_presetting, in2 := 56)
      S_Coil( "Flag".M_FN_03 )
   END_RUNG
   RUNG wire#w1
      { S7_Templates := "SrcType := Int" } EQ_Contact(in1 := "Data".Tempo_presetting, in2 := 60)
      wire#w9
      S_Coil( "Flag".RESET_ALLARM )
   END_RUNG
   RUNG wire#w9
      S_Coil( "Flag".M_FN_06 )
   END_RUNG
   RUNG wire#w1
      { S7_Templates := "SrcType := Int" } EQ_Contact(in1 := "Data".Tempo_presetting, in2 := 62)
      wire#w10
      Contact( "OFF" )
      wire#w11
      { S7_GenerateENO := "TRUE" } Move(in := 850, out1 => "Data".TC01_SETPOINT)
   END_RUNG
   RUNG wire#w11
      { S7_GenerateENO := "TRUE" } Move(in := 500, out1 => "Data".TC03_SETPOINT)
   END_RUNG
   RUNG wire#w10
      S_Coil( "Flag".Start_Burner )
   END_RUNG
   RUNG wire#w10
      S_Coil( "Flag".AUTO_BURNER )
   END_RUNG
   RUNG wire#w1
      { S7_Templates := "SrcType := Int" } EQ_Contact(in1 := "Data".Tempo_presetting, in2 := 65)
      R_Coil( "Flag".Auto_ON1 )
   END_RUNG
   // the same network as SCL:
   #_w1 := "ON" AND NOT "Allarm".Emergency_module_fault AND "Flag".Auto_ON1 AND ("Data".Tipo_preset = 2);
   IF #_w1 AND ("Data".Tempo_presetting = 1) THEN
       "Flag".RESET_ALLARM := TRUE;
       "Flag".Maintenance_ON := FALSE;
   END_IF;
   IF #_w1 AND ("Data".Tempo_presetting = 3) THEN
       "Flag".M_VR_03 := TRUE;
       "Flag".M_VR_04 := TRUE;
       "Flag".M_VR_05 := TRUE;
   END_IF;
   IF #_w1 AND ("Data".Tempo_presetting = 6) THEN
       "Flag".M_SC_01 := TRUE;
       "Flag".M_SC_10 := TRUE;
       "Flag".M_SC_11 := TRUE;
   END_IF;
   IF #_w1 AND ("Data".Tempo_presetting = 10) THEN "Flag".M_FN_04 := TRUE; END_IF;
   IF #_w1 AND ("Data".Tempo_presetting = 18) THEN "Flag".M_VS_01 := TRUE; END_IF;
   IF #_w1 AND ("Data".Tempo_presetting = 21) AND "OFF" THEN "Flag".M_MC_05 := TRUE; END_IF;
   IF #_w1 AND ("Data".Tempo_presetting = 24) THEN "Flag".M_MC_04 := TRUE; END_IF;
   IF #_w1 AND ("Data".Tempo_presetting = 27) THEN "Flag".Enable_R2_GATE := TRUE; END_IF;
   IF #_w1 AND ("Data".Tempo_presetting = 30) THEN "Flag".STANDBY_ON := FALSE; END_IF;
   IF #_w1 AND ("Data".Tempo_presetting = 33) THEN "Flag".M_RD_01_FAN := TRUE; END_IF;
   IF #_w1 AND ("Data".Tempo_presetting = 35) THEN
       "Flag".M_RD_01 := TRUE;
       "Data".SET_PERC_FR01 := 25;
   END_IF;
   IF #_w1 AND ("Data".Tempo_presetting = 40) THEN "Flag".Enable_R1_GATE := TRUE; END_IF;
   IF #_w1 AND ("Data".Tempo_presetting = 43) THEN "Flag".M_BC_01 := TRUE; END_IF;
   IF #_w1 AND ("Data".Tempo_presetting = 46) THEN
       "Flag".M_VR_01 := TRUE;
       "Flag".M_VR_02 := TRUE;
       "Flag".M_CH_01 := TRUE;
   END_IF;
   IF #_w1 AND ("Data".Tempo_presetting = 49) THEN
       "Flag".M_FN_01 := TRUE;
       "Data".SET_PERC_VT01 := 35;
   END_IF;
   IF #_w1 AND ("Data".Tempo_presetting = 52) THEN
       "Flag".M_FN_02 := TRUE;
       "Data".Set_Perc_VT02 := 80;
   END_IF;
   IF #_w1 AND ("Data".Tempo_presetting = 56) THEN "Flag".M_FN_03 := TRUE; END_IF;
   IF #_w1 AND ("Data".Tempo_presetting = 60) THEN
       "Flag".RESET_ALLARM := TRUE;
       "Flag".M_FN_06 := TRUE;
   END_IF;
   #_w2 := #_w1 AND ("Data".Tempo_presetting = 62);
   IF #_w2 AND "OFF" THEN
       "Data".TC01_SETPOINT := 850;
       "Data".TC03_SETPOINT := 500;
   END_IF;
   IF #_w2 THEN
       "Flag".Start_Burner := TRUE;
       "Flag".AUTO_BURNER := TRUE;
   END_IF;
   IF #_w1 AND ("Data".Tempo_presetting = 65) THEN "Flag".Auto_ON1 := FALSE; END_IF;
END_REGION

REGION Network 5: Set Points FN01
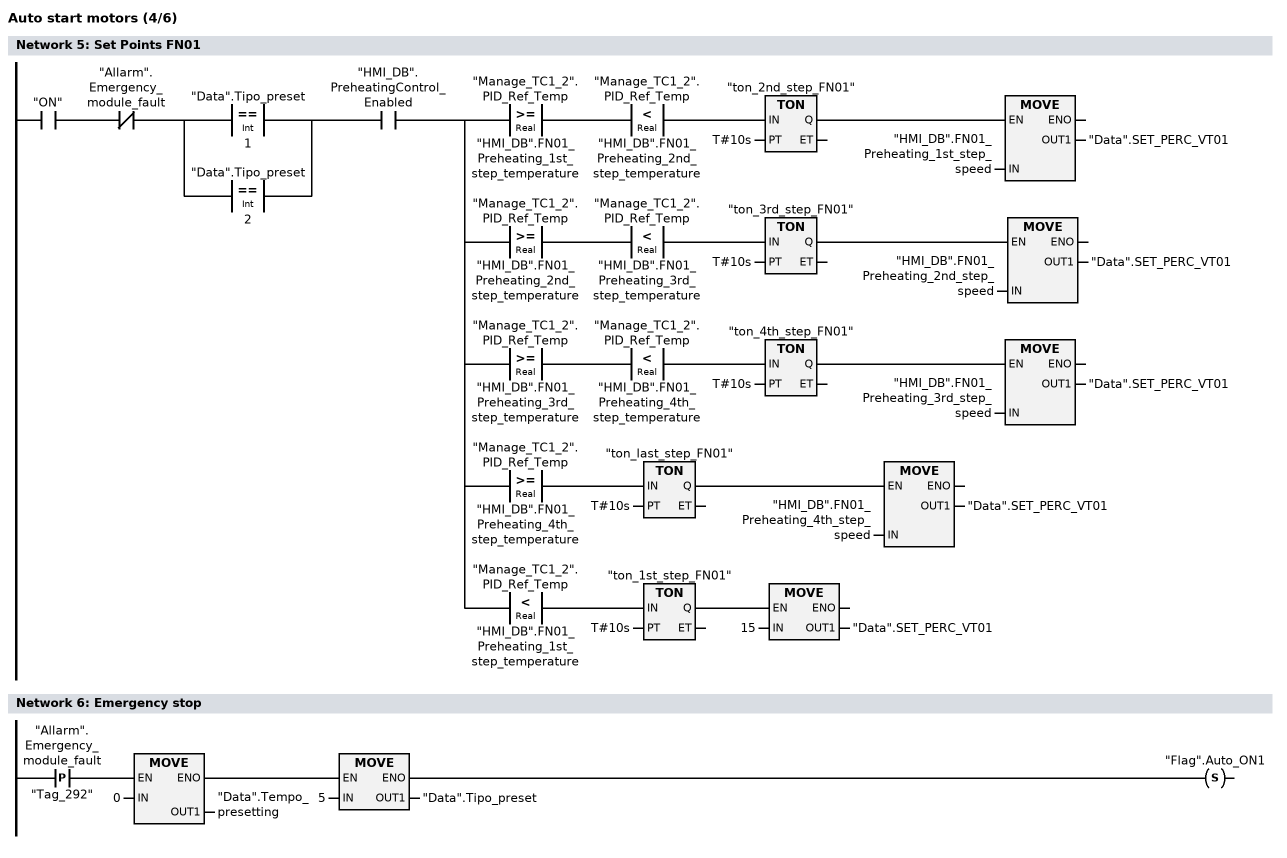
   #_w1 := "ON" AND NOT "Allarm".Emergency_module_fault AND (("Data".Tipo_preset = 1) OR ("Data".Tipo_preset = 2)) AND "HMI_DB".PreheatingControl_Enabled;
   "ton_2nd_step_FN01".TON(IN := #_w1 AND ("Manage_TC1_2".PID_Ref_Temp >= "HMI_DB".FN01_Preheating_1st_step_temperature) AND ("Manage_TC1_2".PID_Ref_Temp < "HMI_DB".FN01_Preheating_2nd_step_temperature),
                           PT := T#10s);
   IF "ton_2nd_step_FN01".Q THEN "Data".SET_PERC_VT01 := "HMI_DB".FN01_Preheating_1st_step_speed; END_IF;
   "ton_3rd_step_FN01".TON(IN := #_w1 AND ("Manage_TC1_2".PID_Ref_Temp >= "HMI_DB".FN01_Preheating_2nd_step_temperature) AND ("Manage_TC1_2".PID_Ref_Temp < "HMI_DB".FN01_Preheating_3rd_step_temperature),
                           PT := T#10s);
   IF "ton_3rd_step_FN01".Q THEN "Data".SET_PERC_VT01 := "HMI_DB".FN01_Preheating_2nd_step_speed; END_IF;
   "ton_4th_step_FN01".TON(IN := #_w1 AND ("Manage_TC1_2".PID_Ref_Temp >= "HMI_DB".FN01_Preheating_3rd_step_temperature) AND ("Manage_TC1_2".PID_Ref_Temp < "HMI_DB".FN01_Preheating_4th_step_temperature),
                           PT := T#10s);
   IF "ton_4th_step_FN01".Q THEN "Data".SET_PERC_VT01 := "HMI_DB".FN01_Preheating_3rd_step_speed; END_IF;
   "ton_last_step_FN01".TON(IN := #_w1 AND ("Manage_TC1_2".PID_Ref_Temp >= "HMI_DB".FN01_Preheating_4th_step_temperature),
                           PT := T#10s);
   IF "ton_last_step_FN01".Q THEN "Data".SET_PERC_VT01 := "HMI_DB".FN01_Preheating_4th_step_speed; END_IF;
   "ton_1st_step_FN01".TON(IN := #_w1 AND ("Manage_TC1_2".PID_Ref_Temp < "HMI_DB".FN01_Preheating_1st_step_temperature),
                           PT := T#10s);
   IF "ton_1st_step_FN01".Q THEN "Data".SET_PERC_VT01 := 15; END_IF;
END_REGION

REGION Network 6: Emergency stop
   RUNG wire#powerrail
      P_Contact(operand := "Allarm".Emergency_module_fault, bit := "Tag_292")
      Move(in := 0, out1 => "Data".Tempo_presetting)
      Move(in := 5, out1 => "Data".Tipo_preset)
      S_Coil( "Flag".Auto_ON1 )
   END_RUNG
   // the same network as SCL:
   #_w1 := "Allarm".Emergency_module_fault AND NOT "Tag_292";   // rising edge of "Allarm".Emergency_module_fault
   "Tag_292" := "Allarm".Emergency_module_fault;
   IF #_w1 THEN
       "Data".Tempo_presetting := 0;
       "Data".Tipo_preset := 5;
       "Flag".Auto_ON1 := TRUE;
   END_IF;
END_REGION

REGION Network 7: Sequenza di presetting 5 : stop motori completo / Presetting sequence 5: complete engine stop
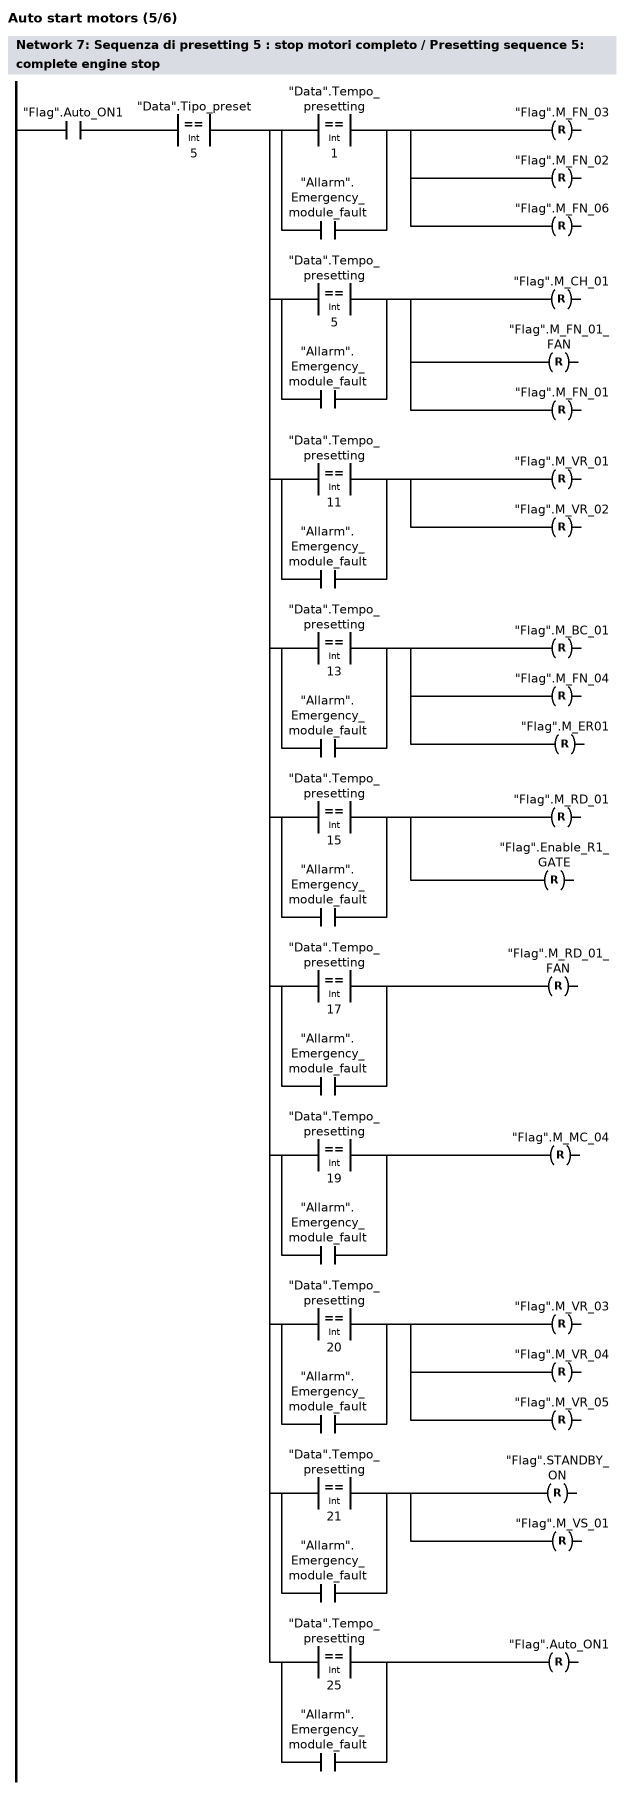
   RUNG wire#powerrail
      Contact( "Flag".Auto_ON1 )
      { S7_Templates := "SrcType := Int" } EQ_Contact(in1 := "Data".Tipo_preset, in2 := 5)
      wire#w1
      { S7_Templates := "SrcType := Int" } EQ_Contact(in1 := "Data".Tempo_presetting, in2 := 1)
      wire#w2
      R_Coil( "Flag".M_FN_03 )
   END_RUNG
   RUNG wire#w1
      Contact( "Allarm".Emergency_module_fault )
   END_RUNG wire#w2
   RUNG wire#w2
      R_Coil( "Flag".M_FN_02 )
   END_RUNG
   RUNG wire#w2
      R_Coil( "Flag".M_FN_06 )
   END_RUNG
   RUNG wire#w1
      { S7_Templates := "SrcType := Int" } EQ_Contact(in1 := "Data".Tempo_presetting, in2 := 5)
      wire#w3
      R_Coil( "Flag".M_CH_01 )
   END_RUNG
   RUNG wire#w1
      Contact( "Allarm".Emergency_module_fault )
   END_RUNG wire#w3
   RUNG wire#w3
      R_Coil( "Flag".M_FN_01_FAN )
   END_RUNG
   RUNG wire#w3
      R_Coil( "Flag".M_FN_01 )
   END_RUNG
   RUNG wire#w1
      { S7_Templates := "SrcType := Int" } EQ_Contact(in1 := "Data".Tempo_presetting, in2 := 11)
      wire#w4
      R_Coil( "Flag".M_VR_01 )
   END_RUNG
   RUNG wire#w1
      Contact( "Allarm".Emergency_module_fault )
   END_RUNG wire#w4
   RUNG wire#w4
      R_Coil( "Flag".M_VR_02 )
   END_RUNG
   RUNG wire#w1
      { S7_Templates := "SrcType := Int" } EQ_Contact(in1 := "Data".Tempo_presetting, in2 := 13)
      wire#w5
      R_Coil( "Flag".M_BC_01 )
   END_RUNG
   RUNG wire#w1
      Contact( "Allarm".Emergency_module_fault )
   END_RUNG wire#w5
   RUNG wire#w5
      R_Coil( "Flag".M_FN_04 )
   END_RUNG
   RUNG wire#w5
      R_Coil( "Flag".M_ER01 )
   END_RUNG
   RUNG wire#w1
      { S7_Templates := "SrcType := Int" } EQ_Contact(in1 := "Data".Tempo_presetting, in2 := 15)
      wire#w6
      R_Coil( "Flag".M_RD_01 )
   END_RUNG
   RUNG wire#w1
      Contact( "Allarm".Emergency_module_fault )
   END_RUNG wire#w6
   RUNG wire#w6
      R_Coil( "Flag".Enable_R1_GATE )
   END_RUNG
   RUNG wire#w1
      { S7_Templates := "SrcType := Int" } EQ_Contact(in1 := "Data".Tempo_presetting, in2 := 17)
      wire#w7
      R_Coil( "Flag".M_RD_01_FAN )
   END_RUNG
   RUNG wire#w1
      Contact( "Allarm".Emergency_module_fault )
   END_RUNG wire#w7
   RUNG wire#w1
      { S7_Templates := "SrcType := Int" } EQ_Contact(in1 := "Data".Tempo_presetting, in2 := 19)
      wire#w8
      R_Coil( "Flag".M_MC_04 )
   END_RUNG
   RUNG wire#w1
      Contact( "Allarm".Emergency_module_fault )
   END_RUNG wire#w8
   RUNG wire#w1
      { S7_Templates := "SrcType := Int" } EQ_Contact(in1 := "Data".Tempo_presetting, in2 := 20)
      wire#w9
      R_Coil( "Flag".M_VR_03 )
   END_RUNG
   RUNG wire#w1
      Contact( "Allarm".Emergency_module_fault )
   END_RUNG wire#w9
   RUNG wire#w9
      R_Coil( "Flag".M_VR_04 )
   END_RUNG
   RUNG wire#w9
      R_Coil( "Flag".M_VR_05 )
   END_RUNG
   RUNG wire#w1
      { S7_Templates := "SrcType := Int" } EQ_Contact(in1 := "Data".Tempo_presetting, in2 := 21)
      wire#w10
      R_Coil( "Flag".STANDBY_ON )
   END_RUNG
   RUNG wire#w1
      Contact( "Allarm".Emergency_module_fault )
   END_RUNG wire#w10
   RUNG wire#w10
      R_Coil( "Flag".M_VS_01 )
   END_RUNG
   RUNG wire#w1
      { S7_Templates := "SrcType := Int" } EQ_Contact(in1 := "Data".Tempo_presetting, in2 := 25)
      wire#w11
      R_Coil( "Flag".Auto_ON1 )
   END_RUNG
   RUNG wire#w1
      Contact( "Allarm".Emergency_module_fault )
   END_RUNG wire#w11
   // the same network as SCL:
   #_w1 := "Flag".Auto_ON1 AND ("Data".Tipo_preset = 5);
   IF #_w1 AND (("Data".Tempo_presetting = 1) OR "Allarm".Emergency_module_fault) THEN
       "Flag".M_FN_03 := FALSE;
       "Flag".M_FN_02 := FALSE;
       "Flag".M_FN_06 := FALSE;
   END_IF;
   IF #_w1 AND (("Data".Tempo_presetting = 5) OR "Allarm".Emergency_module_fault) THEN
       "Flag".M_CH_01 := FALSE;
       "Flag".M_FN_01_FAN := FALSE;
       "Flag".M_FN_01 := FALSE;
   END_IF;
   IF #_w1 AND (("Data".Tempo_presetting = 11) OR "Allarm".Emergency_module_fault) THEN
       "Flag".M_VR_01 := FALSE;
       "Flag".M_VR_02 := FALSE;
   END_IF;
   IF #_w1 AND (("Data".Tempo_presetting = 13) OR "Allarm".Emergency_module_fault) THEN
       "Flag".M_BC_01 := FALSE;
       "Flag".M_FN_04 := FALSE;
       "Flag".M_ER01 := FALSE;
   END_IF;
   IF #_w1 AND (("Data".Tempo_presetting = 15) OR "Allarm".Emergency_module_fault) THEN
       "Flag".M_RD_01 := FALSE;
       "Flag".Enable_R1_GATE := FALSE;
   END_IF;
   IF #_w1 AND (("Data".Tempo_presetting = 17) OR "Allarm".Emergency_module_fault) THEN
       "Flag".M_RD_01_FAN := FALSE;
   END_IF;
   IF #_w1 AND (("Data".Tempo_presetting = 19) OR "Allarm".Emergency_module_fault) THEN
       "Flag".M_MC_04 := FALSE;
   END_IF;
   IF #_w1 AND (("Data".Tempo_presetting = 20) OR "Allarm".Emergency_module_fault) THEN
       "Flag".M_VR_03 := FALSE;
       "Flag".M_VR_04 := FALSE;
       "Flag".M_VR_05 := FALSE;
   END_IF;
   IF #_w1 AND (("Data".Tempo_presetting = 21) OR "Allarm".Emergency_module_fault) THEN
       "Flag".STANDBY_ON := FALSE;
       "Flag".M_VS_01 := FALSE;
   END_IF;
   IF #_w1 AND (("Data".Tempo_presetting = 25) OR "Allarm".Emergency_module_fault) THEN
       "Flag".Auto_ON1 := FALSE;
   END_IF;
END_REGION

REGION Network 8: Sequenza di presetting 6 : nessuna sequenza / Presetting sequence 6: no sequence
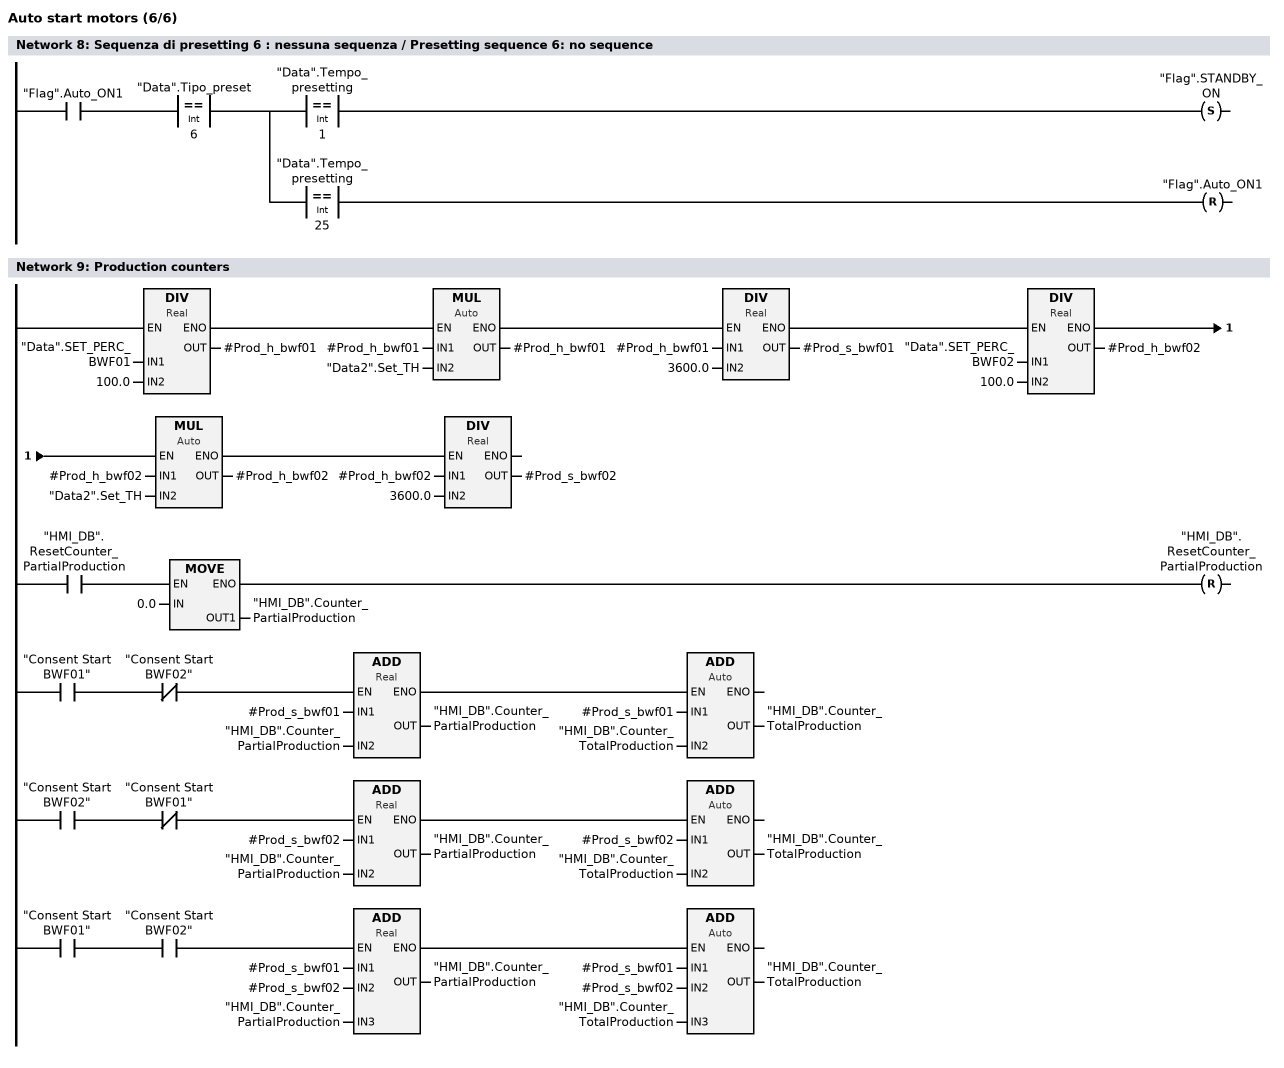
   RUNG wire#powerrail
      Contact( "Flag".Auto_ON1 )
      { S7_Templates := "SrcType := Int" } EQ_Contact(in1 := "Data".Tipo_preset, in2 := 6)
      wire#w1
      { S7_Templates := "SrcType := Int" } EQ_Contact(in1 := "Data".Tempo_presetting, in2 := 1)
      S_Coil( "Flag".STANDBY_ON )
   END_RUNG
   RUNG wire#w1
      { S7_Templates := "SrcType := Int" } EQ_Contact(in1 := "Data".Tempo_presetting, in2 := 25)
      R_Coil( "Flag".Auto_ON1 )
   END_RUNG
   // the same network as SCL:
   #_w1 := "Flag".Auto_ON1 AND ("Data".Tipo_preset = 6);
   IF #_w1 AND ("Data".Tempo_presetting = 1) THEN "Flag".STANDBY_ON := TRUE; END_IF;
   IF #_w1 AND ("Data".Tempo_presetting = 25) THEN "Flag".Auto_ON1 := FALSE; END_IF;
END_REGION

REGION Network 9: Production counters
   RUNG wire#powerrail
      { S7_Templates := "SrcType := Real" } Div(in1 := "Data".SET_PERC_BWF01, in2 := 100.0, out => #Prod_h_bwf01)
      Mul(in1 := #Prod_h_bwf01, in2 := "Data2".Set_TH, out => #Prod_h_bwf01)
      { S7_Templates := "SrcType := Real" } Div(in1 := #Prod_h_bwf01, in2 := 3600.0, out => #Prod_s_bwf01)
      { S7_Templates := "SrcType := Real" } Div(in1 := "Data".SET_PERC_BWF02, in2 := 100.0, out => #Prod_h_bwf02)
      Mul(in1 := #Prod_h_bwf02, in2 := "Data2".Set_TH, out => #Prod_h_bwf02)
      { S7_Templates := "SrcType := Real" } Div(in1 := #Prod_h_bwf02, in2 := 3600.0, out => #Prod_s_bwf02)
   END_RUNG
   RUNG wire#powerrail
      Contact( "HMI_DB".ResetCounter_PartialProduction )
      Move(in := 0.0, out1 => "HMI_DB".Counter_PartialProduction)
      R_Coil( "HMI_DB".ResetCounter_PartialProduction )
   END_RUNG
   RUNG wire#powerrail
      Contact( "Consent Start BWF01" )
      I_Contact( "Consent Start BWF02" )
      { S7_Templates := "SrcType := Real" } Add(in1 := #Prod_s_bwf01, in2 := "HMI_DB".Counter_PartialProduction, out => "HMI_DB".Counter_PartialProduction)
      Add(in1 := #Prod_s_bwf01, in2 := "HMI_DB".Counter_TotalProduction, out => "HMI_DB".Counter_TotalProduction)
   END_RUNG
   RUNG wire#powerrail
      Contact( "Consent Start BWF02" )
      I_Contact( "Consent Start BWF01" )
      { S7_Templates := "SrcType := Real" } Add(in1 := #Prod_s_bwf02, in2 := "HMI_DB".Counter_PartialProduction, out => "HMI_DB".Counter_PartialProduction)
      Add(in1 := #Prod_s_bwf02, in2 := "HMI_DB".Counter_TotalProduction, out => "HMI_DB".Counter_TotalProduction)
   END_RUNG
   RUNG wire#powerrail
      Contact( "Consent Start BWF01" )
      Contact( "Consent Start BWF02" )
      { S7_Templates := "SrcType := Real" } Add(in1 := #Prod_s_bwf01, in2 := #Prod_s_bwf02, in3 := "HMI_DB".Counter_PartialProduction, out => "HMI_DB".Counter_PartialProduction)
      Add(in1 := #Prod_s_bwf01, in2 := #Prod_s_bwf02, in3 := "HMI_DB".Counter_TotalProduction, out => "HMI_DB".Counter_TotalProduction)
   END_RUNG
   // the same network as SCL:
   #Prod_h_bwf01 := "Data".SET_PERC_BWF01 / 100.0;
   #Prod_h_bwf01 := #Prod_h_bwf01 * "Data2".Set_TH;
   #Prod_s_bwf01 := #Prod_h_bwf01 / 3600.0;
   #Prod_h_bwf02 := "Data".SET_PERC_BWF02 / 100.0;
   #Prod_h_bwf02 := #Prod_h_bwf02 * "Data2".Set_TH;
   #Prod_s_bwf02 := #Prod_h_bwf02 / 3600.0;
   IF "HMI_DB".ResetCounter_PartialProduction THEN
       "HMI_DB".Counter_PartialProduction := 0.0;
       "HMI_DB".ResetCounter_PartialProduction := FALSE;
   END_IF;
   IF "Consent Start BWF01" AND NOT "Consent Start BWF02" THEN
       "HMI_DB".Counter_PartialProduction := #Prod_s_bwf01 + "HMI_DB".Counter_PartialProduction;
       "HMI_DB".Counter_TotalProduction := #Prod_s_bwf01 + "HMI_DB".Counter_TotalProduction;
   END_IF;
   IF "Consent Start BWF02" AND NOT "Consent Start BWF01" THEN
       "HMI_DB".Counter_PartialProduction := #Prod_s_bwf02 + "HMI_DB".Counter_PartialProduction;
       "HMI_DB".Counter_TotalProduction := #Prod_s_bwf02 + "HMI_DB".Counter_TotalProduction;
   END_IF;
   IF "Consent Start BWF01" AND "Consent Start BWF02" THEN
       "HMI_DB".Counter_PartialProduction := #Prod_s_bwf01 + #Prod_s_bwf02 + "HMI_DB".Counter_PartialProduction;
       "HMI_DB".Counter_TotalProduction := #Prod_s_bwf01 + #Prod_s_bwf02 + "HMI_DB".Counter_TotalProduction;
   END_IF;
END_REGION
END_FUNCTION

FUNCTION "Signal linearization" : Void   // FC63, LAD
TITLE = Signal linearization
{ S7_Optimized_Access := 'FALSE' }
VERSION : 0.1
   VAR_INPUT
      IN0 : Bool;
      Analog_input : Int;
      Coeff : Int;
      Zero : Int;
   END_VAR
   VAR_OUTPUT
      OutValue : Int;
      Out_of_range : Bool;
   END_VAR
   VAR_TEMP
      App1 : Int;
      App2 : DInt;
      App3 : DInt;
      App4 : DInt;
      App5 : DInt;
      App6 : DInt;
   END_VAR
   VAR_TEMP   // added for the SCL form of the ladder/FBD networks
      _w1 : Bool;
   END_VAR
BEGIN

REGION Network 1
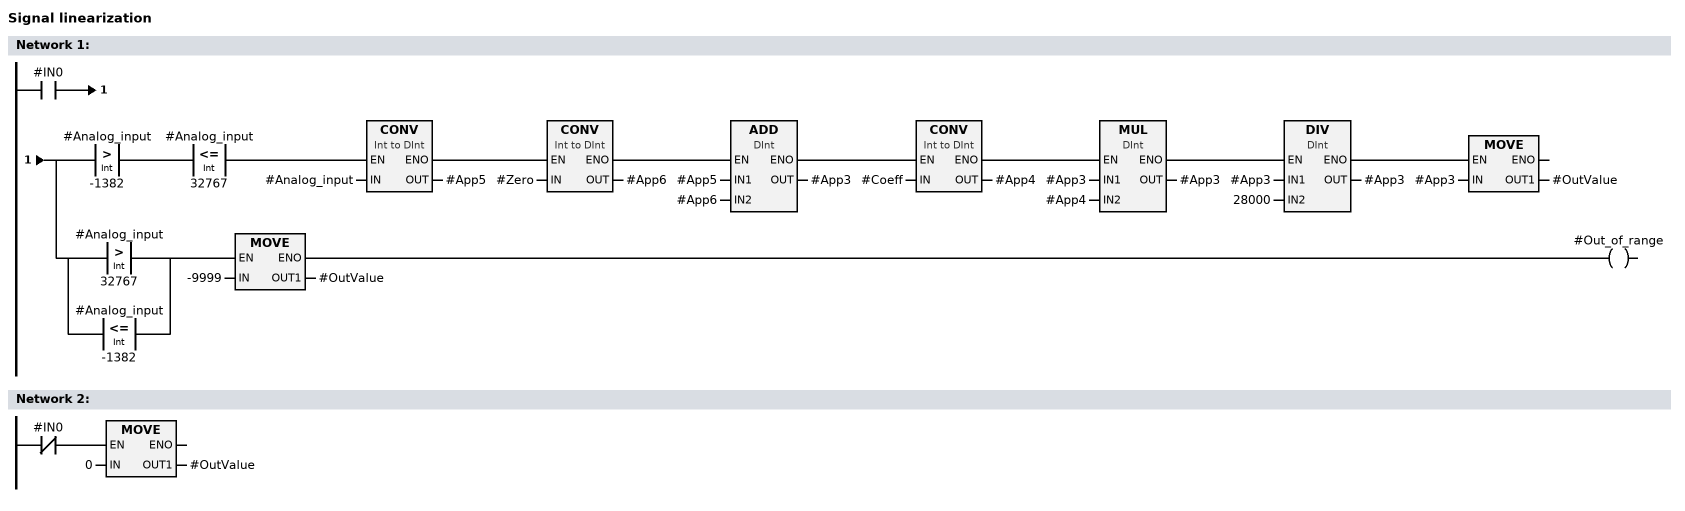
   RUNG wire#powerrail
      Contact( #IN0 )
      wire#w1
      { S7_Templates := "SrcType := Int" } GT_Contact(in1 := #Analog_input, in2 := -1382)
      { S7_Templates := "SrcType := Int" } LE_Contact(in1 := #Analog_input, in2 := 32767)
      { S7_Templates := "[SrcType := Int, DestType := DInt]"; S7_GenerateENO := "TRUE" } Convert(in := #Analog_input, out => #App5)
      { S7_Templates := "[SrcType := Int, DestType := DInt]"; S7_GenerateENO := "TRUE" } Convert(in := #Zero, out => #App6)
      { S7_Templates := "SrcType := DInt"; S7_GenerateENO := "TRUE" } Add(in1 := #App5, in2 := #App6, out => #App3)
      { S7_Templates := "[SrcType := Int, DestType := DInt]"; S7_GenerateENO := "TRUE" } Convert(in := #Coeff, out => #App4)
      { S7_Templates := "SrcType := DInt"; S7_GenerateENO := "TRUE" } Mul(in1 := #App3, in2 := #App4, out => #App3)
      { S7_Templates := "SrcType := DInt"; S7_GenerateENO := "TRUE" } Div(in1 := #App3, in2 := 28000, out => #App3)
      { S7_GenerateENO := "TRUE" } Move(in := #App3, out1 => #OutValue)
   END_RUNG
   RUNG wire#w1
      { S7_Templates := "SrcType := Int" } GT_Contact(in1 := #Analog_input, in2 := 32767)
      wire#w2
      { S7_GenerateENO := "TRUE" } Move(in := -9999, out1 => #OutValue)
      Coil( #Out_of_range )
   END_RUNG
   RUNG wire#w1
      { S7_Templates := "SrcType := Int" } LE_Contact(in1 := #Analog_input, in2 := -1382)
   END_RUNG wire#w2
   // the same network as SCL:
   // ENO of a box is taken as its EN; it also drops when the box reports an error
   IF #IN0 AND (#Analog_input > (-1382)) AND (#Analog_input <= 32767) THEN
       #App5 := INT_TO_DINT(#Analog_input);
       #App6 := INT_TO_DINT(#Zero);
       #App3 := #App5 + #App6;
       #App4 := INT_TO_DINT(#Coeff);
       #App3 := #App3 * #App4;
       #App3 := #App3 / 28000;
       #OutValue := #App3;
   END_IF;
   #_w1 := #IN0 AND ((#Analog_input > 32767) OR (#Analog_input <= (-1382)));
   IF #_w1 THEN #OutValue := -9999; END_IF;
   #Out_of_range := #_w1;
END_REGION

REGION Network 2
   RUNG wire#powerrail
      I_Contact( #IN0 )
      { S7_GenerateENO := "TRUE" } Move(in := 0, out1 => #OutValue)
   END_RUNG
   // the same network as SCL:
   IF NOT #IN0 THEN #OutValue := 0; END_IF;
END_REGION
END_FUNCTION

FUNCTION "R1 scraps gate 2" : Void   // FC99, LAD
TITLE = R1 gate and hydraulic pistons
{ S7_Optimized_Access := 'FALSE' }
VERSION : 0.1
   VAR_TEMP
      PV01_A_TIME : Time;
   END_VAR
   VAR_TEMP   // added for the SCL form of the ladder/FBD networks
      _w1 : Bool;
      _w2 : Bool;
      _w3 : Bool;
      _w4 : Bool;
      _w5 : Bool;
      _w6 : Bool;
      _w7 : Bool;
   END_VAR
BEGIN

REGION Network 1: PV-01
